KUKA KRL program: ps_ltc_geo_c2_Bolha.src, ps_ltc_geo_c2_Bolha.dat

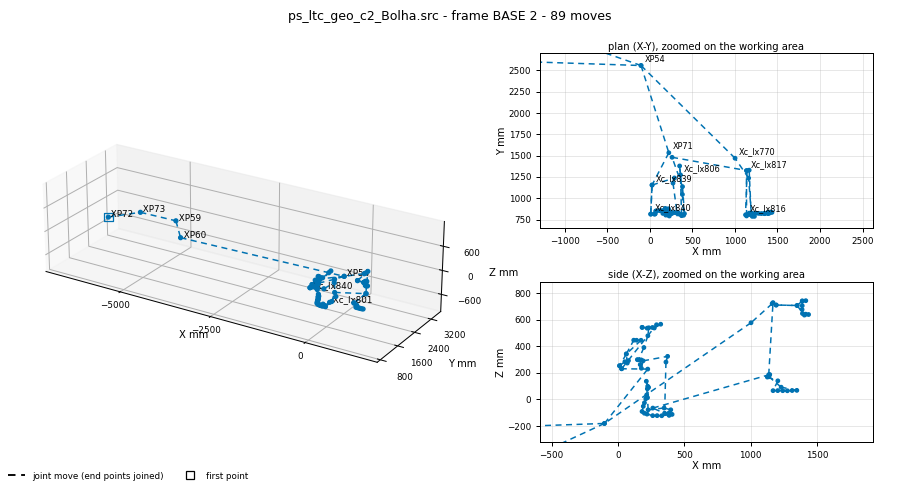
[picture p0: tool path of ps_ltc_geo_c2_Bolha.src in frame BASE 2, 89 of 89 moves have a stored position in this frame; points joined in program order, loops and branches not executed]
--- ps_ltc_geo_c2_Bolha.src ---
&ACCESS RVO1
&REL 11
&COMMENT Solda GUN C2 Geometria
&PARAM DISKPATH = KRC:\R1\Program\SOLDA LTC
DEF ps_ltc_geo_c2_Bolha( )
;FOLD INI
;FOLD SPOTTECH INI
USERSPOT(#INIT)
;ENDFOLD (SPOTTECH INI)
  ;FOLD USER INI
    ;Make your modifications here

  ;ENDFOLD (USER INI)
;ENDFOLD (INI)

; Caracterização dos meios de produção:
; Versão Atual: 03/11/2017
; Changes: Accelo Bolha
; Name: P13.050-R4


chk_w2_wechs_ok ( )     ; CHECK FERRAMENTA: C2

if MaxStandMenge (2) then
  MaxStandmengeErreicht (2)
endif

IF (NOT(GHOST())) THEN
if Elektrodenwechsel (2) then
  e_fraes2()
endif
ENDIF

;FOLD PTP P72 Vel=100 % PDAT95 Tool[2]:GUN C2 Base[2]:ACCELO;%{PE}%R 8.2.20,%MKUKATPBASIS,%CMOVE,%VPTP,%P 1:PTP, 2:P72, 3:, 5:100, 7:PDAT95
$BWDSTART=FALSE
PDAT_ACT=PPDAT95
FDAT_ACT=FP72
BAS(#PTP_PARAMS,100)
PTP XP72
;ENDFOLD
;FOLD PTP P73 CONT Vel=100 % PDAT96 Tool[2]:GUN C2 Base[2]:ACCELO;%{PE}%R 8.2.20,%MKUKATPBASIS,%CMOVE,%VPTP,%P 1:PTP, 2:P73, 3:C_DIS, 5:100, 7:PDAT96
$BWDSTART=FALSE
PDAT_ACT=PPDAT96
FDAT_ACT=FP73
BAS(#PTP_PARAMS,100)
PTP XP73 C_DIS
;ENDFOLD
;FOLD PTP P59 CONT Vel=100 % PDAT79 Tool[2]:GUN C2 Base[2]:ACCELO;%{PE}%R 8.2.20,%MKUKATPBASIS,%CMOVE,%VPTP,%P 1:PTP, 2:P59, 3:C_DIS, 5:100, 7:PDAT79
$BWDSTART=FALSE
PDAT_ACT=PPDAT79
FDAT_ACT=FP59
BAS(#PTP_PARAMS,100)
PTP XP59 C_DIS
;ENDFOLD
;FOLD PTP P60 CONT Vel=100 % PDAT80 Tool[2]:GUN C2 Base[2]:ACCELO;%{PE}%R 8.2.20,%MKUKATPBASIS,%CMOVE,%VPTP,%P 1:PTP, 2:P60, 3:C_DIS, 5:100, 7:PDAT80
$BWDSTART=FALSE
PDAT_ACT=PPDAT80
FDAT_ACT=FP60
BAS(#PTP_PARAMS,100)
PTP XP60 C_DIS
;ENDFOLD
;FOLD PTP P54 CONT Vel=100 % PDAT74 Tool[2]:GUN C2 Base[2]:ACCELO;%{PE}%R 8.2.20,%MKUKATPBASIS,%CMOVE,%VPTP,%P 1:PTP, 2:P54, 3:C_DIS, 5:100, 7:PDAT74
$BWDSTART=FALSE
PDAT_ACT=PPDAT74
FDAT_ACT=FP54
BAS(#PTP_PARAMS,100)
PTP XP54 C_DIS
;ENDFOLD


;FOLD OUT 3339 'R4 soldando' State=TRUE ;%{PE}%R 8.2.20,%MKUKATPBASIS,%COUT,%VOUTX,%P 2:3339, 3:R4 soldando, 5:TRUE, 6:
$OUT[3339]=TRUE
;ENDFOLD
;FOLD WAIT FOR ( IN 3339 'Aguarda lib solsar geometria' );%{PE}%R 8.2.20,%MKUKATPBASIS,%CEXT_WAIT_FOR,%VEXT_WAIT_FOR,%P 2:, 4:, 5:$IN, 6:3339, 7:Aguarda lib solsar geometria, 9:
WAIT FOR  ( $IN[3339] )
;ENDFOLD
;FOLD OUT 3339 'R4 soldando' State=FALSE ;%{PE}%R 8.2.20,%MKUKATPBASIS,%COUT,%VOUTX,%P 2:3339, 3:R4 soldando, 5:FALSE, 6:
$OUT[3339]=FALSE
;ENDFOLD
;FOLD OUT 3348 'Fora area GEOBOX' State=FALSE ;%{PE}%R 8.2.20,%MKUKATPBASIS,%COUT,%VOUTX,%P 2:3348, 3:Fora area GEOBOX, 5:FALSE, 6:
$OUT[3348]=FALSE
;ENDFOLD

;FOLD Collision.Monitoring_AREA_2_On ;%{PE}%MKUKATPUSER
COLLSTOP( 8, 1 ) ;not Interrupt-Controlled
;ENDFOLD


;FOLD PTP P71 CONT Vel=100 % PDAT94 Tool[2]:GUN C2 Base[2]:ACCELO;%{PE}%R 8.2.20,%MKUKATPBASIS,%CMOVE,%VPTP,%P 1:PTP, 2:P71, 3:C_DIS, 5:100, 7:PDAT94
$BWDSTART=FALSE
PDAT_ACT=PPDAT94
FDAT_ACT=FP71
BAS(#PTP_PARAMS,100)
PTP XP71 C_DIS
;ENDFOLD
;FOLD PTP c_lx839 CONT Vel=100 % P_OLP100 Tool[2]:GUN C2 Base[2]:ACCELO;%{PE}%R 8.2.20,%MKUKATPBASIS,%CMOVE,%VPTP,%P 1:PTP, 2:c_lx839, 3:C_DIS, 5:100, 7:P_OLP100
$BWDSTART=FALSE
PDAT_ACT=PP_OLP100
FDAT_ACT=Fc_lx839
BAS(#PTP_PARAMS,100)
PTP Xc_lx839 C_DIS
;ENDFOLD
;FOLD PTP c_lx840 CONT Vel=100 % P_OLP101 Tool[2]:GUN C2 Base[2]:ACCELO;%{PE}%R 8.2.20,%MKUKATPBASIS,%CMOVE,%VPTP,%P 1:PTP, 2:c_lx840, 3:C_DIS, 5:100, 7:P_OLP101
$BWDSTART=FALSE
PDAT_ACT=PP_OLP101
FDAT_ACT=Fc_lx840
BAS(#PTP_PARAMS,100)
PTP Xc_lx840 C_DIS
;ENDFOLD
;FOLD PTP P61 CONT Vel=100 % PDAT81 Tool[2]:GUN C2 Base[2]:ACCELO;%{PE}%R 8.2.20,%MKUKATPBASIS,%CMOVE,%VPTP,%P 1:PTP, 2:P61, 3:C_DIS, 5:100, 7:PDAT81
$BWDSTART=FALSE
PDAT_ACT=PPDAT81
FDAT_ACT=FP61
BAS(#PTP_PARAMS,100)
PTP XP61 C_DIS
;ENDFOLD

;FOLD ; swp_60_0220;%{PE}%R 8.2.20,%MKUKATPBASIS,%CCOMMENT,%VNORMAL,%P 2:swp_60_0220
;ENDFOLD
;FOLD PTP swp_60_0220 PDAT82 SPOT Gun=2 RETR CLS PGNO1=111 ACTIVE=1 Tool[2]:GUN C2 Base[2]:ACCELO;%{PE}%R 8.2.2,%MKUKATPSPOT,%CSPOT,%VPTP,%P 1:PTP, 2:swp_60_0220, 3:, 5:100, 7:PDAT82, 10:2, 12:#FIRST, 14:#CLO, 16:152, 18:1, 20:1, 22:0, 24:1, 25:S_OLP2
$BWDSTART=FALSE
PDAT_ACT=PPDAT82
FDAT_ACT=Fswp_60_0220
BAS(#PTP_PARAMS,PPDAT82.VEL)
S_ACT.GUN=2
S_ACT.PAIR=SDEFAULT.PAIR
S_ACT.RETR=#CLO
S_ACT.CLO_TM=1
S_ACT.PGNO1=111
S_ACT.PGNO2=SDEFAULT.PGNO2
S_ACT.PRESS1=SDEFAULT.PRESS1
S_ACT.PRESS2=SDEFAULT.PRESS2
S_READY=FALSE
PTP Xswp_60_0220
USERSPOT(#SPOT, S_ACT)
WAIT FOR S_READY
;ENDFOLD

;FOLD ; swp_60_0218;%{PE}%R 8.2.20,%MKUKATPBASIS,%CCOMMENT,%VNORMAL,%P 2:swp_60_0218
;ENDFOLD
;FOLD PTP swp_60_0218 PDAT83 SPOT Gun=2 RETR OPN PGNO1=112 ACTIVE=1 Tool[2]:GUN C2 Base[2]:ACCELO;%{PE}%R 8.2.2,%MKUKATPSPOT,%CSPOT,%VPTP,%P 1:PTP, 2:swp_60_0218, 3:, 5:100, 7:PDAT83, 10:2, 12:#FIRST, 14:#OPN, 16:153, 18:1, 20:1, 22:0, 24:1, 25:S_OLP3
$BWDSTART=FALSE
PDAT_ACT=PPDAT83
FDAT_ACT=Fswp_60_0218
BAS(#PTP_PARAMS,PPDAT83.VEL)
S_ACT.GUN=2
S_ACT.PAIR=SDEFAULT.PAIR
S_ACT.RETR=#OPN
S_ACT.CLO_TM=1
S_ACT.PGNO1=112
S_ACT.PGNO2=SDEFAULT.PGNO2
S_ACT.PRESS1=SDEFAULT.PRESS1
S_ACT.PRESS2=SDEFAULT.PRESS2
S_READY=FALSE
PTP Xswp_60_0218
USERSPOT(#SPOT, S_ACT)
WAIT FOR S_READY
;ENDFOLD

;FOLD PTP P62 CONT Vel=100 % PDAT84 Tool[2]:GUN C2 Base[2]:ACCELO;%{PE}%R 8.2.20,%MKUKATPBASIS,%CMOVE,%VPTP,%P 1:PTP, 2:P62, 3:C_DIS, 5:100, 7:PDAT84
$BWDSTART=FALSE
PDAT_ACT=PPDAT84
FDAT_ACT=FP62
BAS(#PTP_PARAMS,100)
PTP XP62 C_DIS
;ENDFOLD

;FOLD ; swp_60_0212;%{PE}%R 8.2.20,%MKUKATPBASIS,%CCOMMENT,%VNORMAL,%P 2:swp_60_0212
;ENDFOLD
;FOLD PTP swp_60_0212 PDAT85 SPOT Gun=2 RETR CLS PGNO1=109 ACTIVE=1 Tool[2]:GUN C2 Base[2]:ACCELO;%{PE}%R 8.2.2,%MKUKATPSPOT,%CSPOT,%VPTP,%P 1:PTP, 2:swp_60_0212, 3:, 5:100, 7:PDAT85, 10:2, 12:#FIRST, 14:#CLO, 16:150, 18:1, 20:0, 22:0, 24:1, 25:NORMAL
$BWDSTART=FALSE
PDAT_ACT=PPDAT85
FDAT_ACT=Fswp_60_0212
BAS(#PTP_PARAMS,PPDAT85.VEL)
S_ACT.GUN=2
S_ACT.PAIR=SDEFAULT.PAIR
S_ACT.RETR=#CLO
S_ACT.CLO_TM=1
S_ACT.PGNO1=109
S_ACT.PGNO2=SDEFAULT.PGNO2
S_ACT.PRESS1=SDEFAULT.PRESS1
S_ACT.PRESS2=SDEFAULT.PRESS2
S_READY=FALSE
PTP Xswp_60_0212
USERSPOT(#SPOT, S_ACT)
WAIT FOR S_READY
;ENDFOLD

;FOLD ; swp_60_0210;%{PE}%R 8.2.20,%MKUKATPBASIS,%CCOMMENT,%VNORMAL,%P 2:swp_60_0210
;ENDFOLD
;FOLD PTP swp_60_0210 PDAT86 SPOT Gun=2 RETR CLS PGNO1=113 ACTIVE=1 Tool[2]:GUN C2 Base[2]:ACCELO;%{PE}%R 8.2.2,%MKUKATPSPOT,%CSPOT,%VPTP,%P 1:PTP, 2:swp_60_0210, 3:, 5:100, 7:PDAT86, 10:2, 12:#FIRST, 14:#CLO, 16:154, 18:1, 20:1, 22:0, 24:1, 25:S_OLP4
$BWDSTART=FALSE
PDAT_ACT=PPDAT86
FDAT_ACT=Fswp_60_0210
BAS(#PTP_PARAMS,PPDAT86.VEL)
S_ACT.GUN=2
S_ACT.PAIR=SDEFAULT.PAIR
S_ACT.RETR=#CLO
S_ACT.CLO_TM=1
S_ACT.PGNO1=113
S_ACT.PGNO2=SDEFAULT.PGNO2
S_ACT.PRESS1=SDEFAULT.PRESS1
S_ACT.PRESS2=SDEFAULT.PRESS2
S_READY=FALSE
PTP Xswp_60_0210
USERSPOT(#SPOT, S_ACT)
WAIT FOR S_READY
;ENDFOLD

;FOLD ; swp_60_0208;%{PE}%R 8.2.20,%MKUKATPBASIS,%CCOMMENT,%VNORMAL,%P 2:swp_60_0208
;ENDFOLD
;FOLD PTP swp_60_0208 PDAT87 SPOT Gun=2 RETR OPN PGNO1=108 ACTIVE=1 Tool[2]:GUN C2 Base[2]:ACCELO;%{PE}%R 8.2.2,%MKUKATPSPOT,%CSPOT,%VPTP,%P 1:PTP, 2:swp_60_0208, 3:, 5:100, 7:PDAT87, 10:2, 12:#FIRST, 14:#OPN, 16:149, 18:1, 20:0, 22:0, 24:1, 25:NORMAL
$BWDSTART=FALSE
PDAT_ACT=PPDAT87
FDAT_ACT=Fswp_60_0208
BAS(#PTP_PARAMS,PPDAT87.VEL)
S_ACT.GUN=2
S_ACT.PAIR=SDEFAULT.PAIR
S_ACT.RETR=#OPN
S_ACT.CLO_TM=1
S_ACT.PGNO1=108
S_ACT.PGNO2=SDEFAULT.PGNO2
S_ACT.PRESS1=SDEFAULT.PRESS1
S_ACT.PRESS2=SDEFAULT.PRESS2
S_READY=FALSE
PTP Xswp_60_0208
USERSPOT(#SPOT, S_ACT)
WAIT FOR S_READY
;ENDFOLD

;FOLD PTP P65 CONT Vel=100 % PDAT88 Tool[2]:GUN C2 Base[2]:ACCELO;%{PE}%R 8.2.20,%MKUKATPBASIS,%CMOVE,%VPTP,%P 1:PTP, 2:P65, 3:C_DIS, 5:100, 7:PDAT88
$BWDSTART=FALSE
PDAT_ACT=PPDAT88
FDAT_ACT=FP65
BAS(#PTP_PARAMS,100)
PTP XP65 C_DIS
;ENDFOLD
;FOLD PTP P66 CONT Vel=100 % PDAT89 Tool[2]:GUN C2 Base[2]:ACCELO;%{PE}%R 8.2.20,%MKUKATPBASIS,%CMOVE,%VPTP,%P 1:PTP, 2:P66, 3:C_DIS, 5:100, 7:PDAT89
$BWDSTART=FALSE
PDAT_ACT=PPDAT89
FDAT_ACT=FP66
BAS(#PTP_PARAMS,100)
PTP XP66 C_DIS
;ENDFOLD
;FOLD PTP P67 CONT Vel=100 % PDAT90 Tool[2]:GUN C2 Base[2]:ACCELO;%{PE}%R 8.2.20,%MKUKATPBASIS,%CMOVE,%VPTP,%P 1:PTP, 2:P67, 3:C_DIS, 5:100, 7:PDAT90
$BWDSTART=FALSE
PDAT_ACT=PPDAT90
FDAT_ACT=FP67
BAS(#PTP_PARAMS,100)
PTP XP67 C_DIS
;ENDFOLD
;FOLD PTP P68 CONT Vel=100 % PDAT91 Tool[2]:GUN C2 Base[2]:ACCELO;%{PE}%R 8.2.20,%MKUKATPBASIS,%CMOVE,%VPTP,%P 1:PTP, 2:P68, 3:C_DIS, 5:100, 7:PDAT91
$BWDSTART=FALSE
PDAT_ACT=PPDAT91
FDAT_ACT=FP68
BAS(#PTP_PARAMS,100)
PTP XP68 C_DIS
;ENDFOLD
;FOLD PTP P69 CONT Vel=100 % PDAT92 Tool[2]:GUN C2 Base[2]:ACCELO;%{PE}%R 8.2.20,%MKUKATPBASIS,%CMOVE,%VPTP,%P 1:PTP, 2:P69, 3:C_DIS, 5:100, 7:PDAT92
$BWDSTART=FALSE
PDAT_ACT=PPDAT92
FDAT_ACT=FP69
BAS(#PTP_PARAMS,100)
PTP XP69 C_DIS
;ENDFOLD
;FOLD PTP c_lx791 CONT Vel=100 % P_OLP29 Tool[2]:GUN C2 Base[2]:ACCELO;%{PE}%R8.2,%MKUKATPBASIS,%CMOVE,%VPTP,%P 1:PTP, 2:c_lx791, 3:C_DIS, 5:100, 7:P_OLP29
$BWDSTART = FALSE
PDAT_ACT= PP_OLP29
FDAT_ACT= Fc_lx791
BAS(#PTP_PARAMS,100)
PTP Xc_lx791 C_DIS
;ENDFOLD
;FOLD PTP c_lx794 CONT Vel=100 % P_OLP30 Tool[2]:GUN C2 Base[2]:ACCELO;%{PE}%R8.2,%MKUKATPBASIS,%CMOVE,%VPTP,%P 1:PTP, 2:c_lx794, 3:C_DIS, 5:100, 7:P_OLP30
$BWDSTART = FALSE
PDAT_ACT= PP_OLP30
FDAT_ACT= Fc_lx794
BAS(#PTP_PARAMS,100)
PTP Xc_lx794 C_DIS
;ENDFOLD
;FOLD PTP P10 CONT Vel=100 % PDAT19 Tool[2]:GUN C2 Base[2]:ACCELO;%{PE}%R 8.2.20,%MKUKATPBASIS,%CMOVE,%VPTP,%P 1:PTP, 2:P10, 3:C_DIS, 5:100, 7:PDAT19
$BWDSTART=FALSE
PDAT_ACT=PPDAT19
FDAT_ACT=FP10
BAS(#PTP_PARAMS,100)
PTP XP10 C_DIS
;ENDFOLD

;FOLD ; swp_60_0202;%{PE}%R 8.2.20,%MKUKATPBASIS,%CCOMMENT,%VNORMAL,%P 2:swp_60_0202
;ENDFOLD
;FOLD PTP swp_60_0202 PDAT29 SPOT Gun=2 RETR CLS PGNO1=110 ACTIVE=1 Tool[2]:GUN C2 Base[2]:ACCELO;%{PE}%R 8.2.2,%MKUKATPSPOT,%CSPOT,%VPTP,%P 1:PTP, 2:swp_60_0202, 3:, 5:100, 7:PDAT29, 10:2, 12:#FIRST, 14:#CLO, 16:151, 18:1, 20:1, 22:0, 24:1, 25:S_OLP1
$BWDSTART=FALSE
PDAT_ACT=PPDAT29
FDAT_ACT=Fswp_60_0202
BAS(#PTP_PARAMS,PPDAT29.VEL)
S_ACT.GUN=2
S_ACT.PAIR=SDEFAULT.PAIR
S_ACT.RETR=#CLO
S_ACT.CLO_TM=1
S_ACT.PGNO1=110
S_ACT.PGNO2=SDEFAULT.PGNO2
S_ACT.PRESS1=SDEFAULT.PRESS1
S_ACT.PRESS2=SDEFAULT.PRESS2
S_READY=FALSE
PTP Xswp_60_0202
USERSPOT(#SPOT, S_ACT)
WAIT FOR S_READY
;ENDFOLD

;FOLD ; swp 60_0204;%{PE}%R 8.2.20,%MKUKATPBASIS,%CCOMMENT,%VNORMAL,%P 2:swp  60_0204
;ENDFOLD
;FOLD PTP swp_60_0204 PDAT44 SPOT Gun=2 RETR OPN PgNo1=107 ACTIVE=1 Tool[2]:GUN C2 Base[2]:ACCELO;%{PE}%R 8.2.2,%MKUKATPSPOT,%CSPOT,%VPTP,%P 1:PTP, 2:swp_60_0204, 3:, 5:100, 7:PDAT44, 10:2, 12:#FIRST, 14:#OPN, 16:107, 18:1, 20:0, 22:0, 24:1, 25:NORMAL
$BWDSTART=FALSE
PDAT_ACT=PPDAT44
FDAT_ACT=Fswp_60_0204
BAS(#PTP_PARAMS,PPDAT44.VEL)
S_ACT.GUN=2
S_ACT.PAIR=SDEFAULT.PAIR
S_ACT.RETR=#OPN
S_ACT.CLO_TM=1
S_ACT.PGNO1=107
S_ACT.PGNO2=SDEFAULT.PGNO2
S_ACT.PRESS1=SDEFAULT.PRESS1
S_ACT.PRESS2=SDEFAULT.PRESS2
S_READY=FALSE
PTP Xswp_60_0204
USERSPOT(#SPOT, S_ACT)
WAIT FOR S_READY
;ENDFOLD

;FOLD PTP P28 CONT Vel=100 % PDAT45 Tool[2]:GUN C2 Base[2]:ACCELO;%{PE}%R 8.2.20,%MKUKATPBASIS,%CMOVE,%VPTP,%P 1:PTP, 2:P28, 3:C_DIS, 5:100, 7:PDAT45
$BWDSTART=FALSE
PDAT_ACT=PPDAT45
FDAT_ACT=FP28
BAS(#PTP_PARAMS,100)
PTP XP28 C_DIS
;ENDFOLD

;FOLD ; swp_60_0206;%{PE}%R 8.2.20,%MKUKATPBASIS,%CCOMMENT,%VNORMAL,%P 2:swp_60_0206
;ENDFOLD
;FOLD PTP swp_60_0206 P_OLP92 SPOT Gun=2 RETR OPN PGNO1=114 ACTIVE=1 Tool[2]:GUN C2 Base[2]:ACCELO;%{PE}%R 8.2.2,%MKUKATPSPOT,%CSPOT,%VPTP,%P 1:PTP, 2:swp_60_0206, 3:, 5:100, 7:P_OLP92, 10:2, 12:#FIRST, 14:#OPN, 16:155, 18:1, 20:1, 22:0, 24:1, 25:S_OLP5
$BWDSTART=FALSE
PDAT_ACT=PP_OLP92
FDAT_ACT=Fswp_60_0206
BAS(#PTP_PARAMS,PP_OLP92.VEL)
S_ACT.GUN=2
S_ACT.PAIR=SDEFAULT.PAIR
S_ACT.RETR=#OPN
S_ACT.CLO_TM=1
S_ACT.PGNO1=114
S_ACT.PGNO2=SDEFAULT.PGNO2
S_ACT.PRESS1=SDEFAULT.PRESS1
S_ACT.PRESS2=SDEFAULT.PRESS2
S_READY=FALSE
PTP Xswp_60_0206
USERSPOT(#SPOT, S_ACT)
WAIT FOR S_READY
;ENDFOLD

;FOLD PTP c_lx836 CONT Vel=100 % P_OLP93 Tool[2]:GUN C2 Base[2]:ACCELO;%{PE}%R 8.2.20,%MKUKATPBASIS,%CMOVE,%VPTP,%P 1:PTP, 2:c_lx836, 3:C_DIS, 5:100, 7:P_OLP93
$BWDSTART=FALSE
PDAT_ACT=PP_OLP93
FDAT_ACT=Fc_lx836
BAS(#PTP_PARAMS,100)
PTP Xc_lx836 C_DIS
;ENDFOLD
;FOLD PTP c_lx837 CONT Vel=100 % P_OLP94 Tool[2]:GUN C2 Base[2]:ACCELO;%{PE}%R 8.2.20,%MKUKATPBASIS,%CMOVE,%VPTP,%P 1:PTP, 2:c_lx837, 3:C_DIS, 5:100, 7:P_OLP94
$BWDSTART=FALSE
PDAT_ACT=PP_OLP94
FDAT_ACT=Fc_lx837
BAS(#PTP_PARAMS,100)
PTP Xc_lx837 C_DIS
;ENDFOLD

;FOLD ; swp_60_0222;%{PE}%R 8.2.20,%MKUKATPBASIS,%CCOMMENT,%VNORMAL,%P 2:swp_60_0222
;ENDFOLD
;FOLD PTP swp_60_0222 P_OLP95 SPOT Gun=2 RETR CLS PGNO1=115 ACTIVE=1 Tool[2]:GUN C2 Base[2]:ACCELO;%{PE}%R 8.2.2,%MKUKATPSPOT,%CSPOT,%VPTP,%P 1:PTP, 2:swp_60_0222, 3:, 5:100, 7:P_OLP95, 10:2, 12:#FIRST, 14:#CLO, 16:156, 18:1, 20:1, 22:0, 24:1, 25:S_OLP6
$BWDSTART=FALSE
PDAT_ACT=PP_OLP95
FDAT_ACT=Fswp_60_0222
BAS(#PTP_PARAMS,PP_OLP95.VEL)
S_ACT.GUN=2
S_ACT.PAIR=SDEFAULT.PAIR
S_ACT.RETR=#CLO
S_ACT.CLO_TM=1
S_ACT.PGNO1=115
S_ACT.PGNO2=SDEFAULT.PGNO2
S_ACT.PRESS1=SDEFAULT.PRESS1
S_ACT.PRESS2=SDEFAULT.PRESS2
S_READY=FALSE
PTP Xswp_60_0222
USERSPOT(#SPOT, S_ACT)
WAIT FOR S_READY
;ENDFOLD

;FOLD PTP c_lx838 CONT Vel=100 % P_OLP96 Tool[2]:GUN C2 Base[2]:ACCELO;%{PE}%R 8.2.20,%MKUKATPBASIS,%CMOVE,%VPTP,%P 1:PTP, 2:c_lx838, 3:C_DIS, 5:100, 7:P_OLP96
$BWDSTART=FALSE
PDAT_ACT=PP_OLP96
FDAT_ACT=Fc_lx838
BAS(#PTP_PARAMS,100)
PTP Xc_lx838 C_DIS
;ENDFOLD

;FOLD ; swp_60_0226;%{PE}%R 8.2.20,%MKUKATPBASIS,%CCOMMENT,%VNORMAL,%P 2:swp_60_0226
;ENDFOLD
;FOLD PTP swp_60_0226 P_OLP97 SPOT Gun=2 RETR CLS PGNO1=116 ACTIVE=1 Tool[2]:GUN C2 Base[2]:ACCELO;%{PE}%R 8.2.2,%MKUKATPSPOT,%CSPOT,%VPTP,%P 1:PTP, 2:swp_60_0226, 3:, 5:100, 7:P_OLP97, 10:2, 12:#FIRST, 14:#CLO, 16:157, 18:1, 20:1, 22:0, 24:1, 25:S_OLP7
$BWDSTART=FALSE
PDAT_ACT=PP_OLP97
FDAT_ACT=Fswp_60_0226
BAS(#PTP_PARAMS,PP_OLP97.VEL)
S_ACT.GUN=2
S_ACT.PAIR=SDEFAULT.PAIR
S_ACT.RETR=#CLO
S_ACT.CLO_TM=1
S_ACT.PGNO1=116
S_ACT.PGNO2=SDEFAULT.PGNO2
S_ACT.PRESS1=SDEFAULT.PRESS1
S_ACT.PRESS2=SDEFAULT.PRESS2
S_READY=FALSE
PTP Xswp_60_0226
USERSPOT(#SPOT, S_ACT)
WAIT FOR S_READY
;ENDFOLD

;FOLD ; swp_60_0230;%{PE}%R 5.4.33,%MKUKATPBASIS,%CCOMMENT,%VNORMAL,%P 2:swp_60_0230
;ENDFOLD
;FOLD PTP swp_60_0230 P_OLP38 SPOT Gun=2 RETR OPN PGNO1=117 ACTIVE=1 Tool[2]:GUN C2 Base[2]:ACCELO;%{PE}%R 8.2.2,%MKUKATPSPOT,%CSPOT,%VPTP,%P 1:PTP, 2:swp_60_0230, 3:, 5:100, 7:P_OLP38, 10:2, 12:#FIRST, 14:#OPN, 16:158, 18:1, 20:1, 22:0, 24:1, 25:S_OLP8
$BWDSTART=FALSE
PDAT_ACT=PP_OLP38
FDAT_ACT=Fswp_60_0230
BAS(#PTP_PARAMS,PP_OLP38.VEL)
S_ACT.GUN=2
S_ACT.PAIR=SDEFAULT.PAIR
S_ACT.RETR=#OPN
S_ACT.CLO_TM=1
S_ACT.PGNO1=117
S_ACT.PGNO2=SDEFAULT.PGNO2
S_ACT.PRESS1=SDEFAULT.PRESS1
S_ACT.PRESS2=SDEFAULT.PRESS2
S_READY=FALSE
PTP Xswp_60_0230
USERSPOT(#SPOT, S_ACT)
WAIT FOR S_READY
;ENDFOLD

;FOLD PTP c_lx803 CONT Vel=100 % P_OLP39 Tool[2]:GUN C2 Base[2]:ACCELO;%{PE}%R8.2,%MKUKATPBASIS,%CMOVE,%VPTP,%P 1:PTP, 2:c_lx803, 3:C_DIS, 5:100, 7:P_OLP39
$BWDSTART = FALSE
PDAT_ACT= PP_OLP39
FDAT_ACT= Fc_lx803
BAS(#PTP_PARAMS,100)
PTP Xc_lx803 C_DIS
;ENDFOLD
;FOLD PTP P26 CONT Vel=100 % PDAT43 Tool[2]:GUN C2 Base[2]:ACCELO;%{PE}%R 8.2.20,%MKUKATPBASIS,%CMOVE,%VPTP,%P 1:PTP, 2:P26, 3:C_DIS, 5:100, 7:PDAT43
$BWDSTART=FALSE
PDAT_ACT=PPDAT43
FDAT_ACT=FP26
BAS(#PTP_PARAMS,100)
PTP XP26 C_DIS
;ENDFOLD
;FOLD PTP c_lx806 CONT Vel=100 % P_OLP42 Tool[2]:GUN C2 Base[2]:ACCELO;%{PE}%R8.2,%MKUKATPBASIS,%CMOVE,%VPTP,%P 1:PTP, 2:c_lx806, 3:C_DIS, 5:100, 7:P_OLP42
$BWDSTART = FALSE
PDAT_ACT= PP_OLP42
FDAT_ACT= Fc_lx806
BAS(#PTP_PARAMS,100)
PTP Xc_lx806 C_DIS
;ENDFOLD
;FOLD PTP c_lx831 Vel=100 % P_OLP86 Tool[2]:GUN C2 Base[2]:ACCELO;%{PE}%R 8.2.20,%MKUKATPBASIS,%CMOVE,%VPTP,%P 1:PTP, 2:c_lx831, 3:, 5:100, 7:P_OLP86
$BWDSTART=FALSE
PDAT_ACT=PP_OLP86
FDAT_ACT=Fc_lx831
BAS(#PTP_PARAMS,100)
PTP Xc_lx831
;ENDFOLD
;FOLD PTP c_lx801 CONT Vel=100 % P_OLP46 Tool[2]:GUN C2 Base[2]:ACCELO;%{PE}%R 8.2.20,%MKUKATPBASIS,%CMOVE,%VPTP,%P 1:PTP, 2:c_lx801, 3:C_DIS, 5:100, 7:P_OLP46
$BWDSTART=FALSE
PDAT_ACT=PP_OLP46
FDAT_ACT=Fc_lx801
BAS(#PTP_PARAMS,100)
PTP Xc_lx801 C_DIS
;ENDFOLD
;FOLD PTP c_lx802 CONT Vel=100 % P_OLP47 Tool[2]:GUN C2 Base[2]:ACCELO;%{PE}%R 8.2.20,%MKUKATPBASIS,%CMOVE,%VPTP,%P 1:PTP, 2:c_lx802, 3:C_DIS, 5:100, 7:P_OLP47
$BWDSTART=FALSE
PDAT_ACT=PP_OLP47
FDAT_ACT=Fc_lx802
BAS(#PTP_PARAMS,100)
PTP Xc_lx802 C_DIS
;ENDFOLD
;FOLD PTP c_lx800 CONT Vel=100 % P_OLP48 Tool[2]:GUN C2 Base[2]:ACCELO;%{PE}%R 8.2.20,%MKUKATPBASIS,%CMOVE,%VPTP,%P 1:PTP, 2:c_lx800, 3:C_DIS, 5:100, 7:P_OLP48
$BWDSTART=FALSE
PDAT_ACT=PP_OLP48
FDAT_ACT=Fc_lx800
BAS(#PTP_PARAMS,100)
PTP Xc_lx800 C_DIS
;ENDFOLD
;FOLD PTP c_lx799 CONT Vel=100 % P_OLP49 Tool[2]:GUN C2 Base[2]:ACCELO;%{PE}%R 8.2.20,%MKUKATPBASIS,%CMOVE,%VPTP,%P 1:PTP, 2:c_lx799, 3:C_DIS, 5:100, 7:P_OLP49
$BWDSTART=FALSE
PDAT_ACT=PP_OLP49
FDAT_ACT=Fc_lx799
BAS(#PTP_PARAMS,100)
PTP Xc_lx799 C_DIS
;ENDFOLD
;FOLD PTP P7 CONT Vel=100 % PDAT16 Tool[2]:GUN C2 Base[2]:ACCELO;%{PE}%R 8.2.20,%MKUKATPBASIS,%CMOVE,%VPTP,%P 1:PTP, 2:P7, 3:C_DIS, 5:100, 7:PDAT16
$BWDSTART=FALSE
PDAT_ACT=PPDAT16
FDAT_ACT=FP7
BAS(#PTP_PARAMS,100)
PTP XP7 C_DIS
;ENDFOLD
;FOLD PTP c_lx798 CONT Vel=100 % P_OLP50 Tool[2]:GUN C2 Base[2]:ACCELO;%{PE}%R 8.2.20,%MKUKATPBASIS,%CMOVE,%VPTP,%P 1:PTP, 2:c_lx798, 3:C_DIS, 5:100, 7:P_OLP50
$BWDSTART=FALSE
PDAT_ACT=PP_OLP50
FDAT_ACT=Fc_lx798
BAS(#PTP_PARAMS,100)
PTP Xc_lx798 C_DIS
;ENDFOLD

;FOLD ; swp_60_0236;%{PE}%R 5.4.33,%MKUKATPBASIS,%CCOMMENT,%VNORMAL,%P 2:swp_60_0236
;ENDFOLD
;FOLD PTP swp_60_0236 P_OLP51 SPOT Gun=2 RETR CLS PGNO1=118 ACTIVE=1 Tool[2]:GUN C2 Base[2]:ACCELO;%{PE}%R 8.2.2,%MKUKATPSPOT,%CSPOT,%VPTP,%P 1:PTP, 2:swp_60_0236, 3:, 5:100, 7:P_OLP51, 10:2, 12:#FIRST, 14:#CLO, 16:159, 18:1, 20:1, 22:0, 24:1, 25:S_OLP9
$BWDSTART=FALSE
PDAT_ACT=PP_OLP51
FDAT_ACT=Fswp_60_0236
BAS(#PTP_PARAMS,PP_OLP51.VEL)
S_ACT.GUN=2
S_ACT.PAIR=SDEFAULT.PAIR
S_ACT.RETR=#CLO
S_ACT.CLO_TM=1
S_ACT.PGNO1=118
S_ACT.PGNO2=SDEFAULT.PGNO2
S_ACT.PRESS1=SDEFAULT.PRESS1
S_ACT.PRESS2=SDEFAULT.PRESS2
S_READY=FALSE
PTP Xswp_60_0236
USERSPOT(#SPOT, S_ACT)
WAIT FOR S_READY
;ENDFOLD

;FOLD ; swp_60_0238;%{PE}%R 8.2.20,%MKUKATPBASIS,%CCOMMENT,%VNORMAL,%P 2:swp_60_0238
;ENDFOLD
;FOLD PTP swp_60_0238 PDAT63 SPOT Gun=2 RETR CLS PGNO1=102 ACTIVE=1 Tool[2]:GUN C2 Base[2]:ACCELO;%{PE}%R 8.2.2,%MKUKATPSPOT,%CSPOT,%VPTP,%P 1:PTP, 2:swp_60_0238, 3:, 5:100, 7:PDAT63, 10:2, 12:#FIRST, 14:#CLO, 16:143, 18:1, 20:0, 22:0, 24:1, 25:NORMAL
$BWDSTART=FALSE
PDAT_ACT=PPDAT63
FDAT_ACT=Fswp_60_0238
BAS(#PTP_PARAMS,PPDAT63.VEL)
S_ACT.GUN=2
S_ACT.PAIR=SDEFAULT.PAIR
S_ACT.RETR=#CLO
S_ACT.CLO_TM=1
S_ACT.PGNO1=102
S_ACT.PGNO2=SDEFAULT.PGNO2
S_ACT.PRESS1=SDEFAULT.PRESS1
S_ACT.PRESS2=SDEFAULT.PRESS2
S_READY=FALSE
PTP Xswp_60_0238
USERSPOT(#SPOT, S_ACT)
WAIT FOR S_READY
;ENDFOLD

;FOLD ; swp_60_0240;%{PE}%R 8.2.20,%MKUKATPBASIS,%CCOMMENT,%VNORMAL,%P 2:swp_60_0240
;ENDFOLD
;FOLD PTP swp_60_0240 PDAT64 SPOT Gun=2 RETR CLS PGNO1=101 ACTIVE=1 Tool[2]:GUN C2 Base[2]:ACCELO;%{PE}%R 8.2.2,%MKUKATPSPOT,%CSPOT,%VPTP,%P 1:PTP, 2:swp_60_0240, 3:, 5:100, 7:PDAT64, 10:2, 12:#FIRST, 14:#CLO, 16:142, 18:1, 20:0, 22:0, 24:1, 25:NORMAL
$BWDSTART=FALSE
PDAT_ACT=PPDAT64
FDAT_ACT=Fswp_60_0240
BAS(#PTP_PARAMS,PPDAT64.VEL)
S_ACT.GUN=2
S_ACT.PAIR=SDEFAULT.PAIR
S_ACT.RETR=#CLO
S_ACT.CLO_TM=1
S_ACT.PGNO1=101
S_ACT.PGNO2=SDEFAULT.PGNO2
S_ACT.PRESS1=SDEFAULT.PRESS1
S_ACT.PRESS2=SDEFAULT.PRESS2
S_READY=FALSE
PTP Xswp_60_0240
USERSPOT(#SPOT, S_ACT)
WAIT FOR S_READY
;ENDFOLD

;FOLD ; swp_60_0242;%{PE}%R 8.2.20,%MKUKATPBASIS,%CCOMMENT,%VNORMAL,%P 2:swp_60_0242
;ENDFOLD
;FOLD PTP swp_60_0242 PDAT65 SPOT Gun=2 RETR CLS PGNO1=100 ACTIVE=1 Tool[2]:GUN C2 Base[2]:ACCELO;%{PE}%R 8.2.2,%MKUKATPSPOT,%CSPOT,%VPTP,%P 1:PTP, 2:swp_60_0242, 3:, 5:100, 7:PDAT65, 10:2, 12:#FIRST, 14:#CLO, 16:141, 18:1, 20:0, 22:0, 24:1, 25:NORMAL
$BWDSTART=FALSE
PDAT_ACT=PPDAT65
FDAT_ACT=Fswp_60_0242
BAS(#PTP_PARAMS,PPDAT65.VEL)
S_ACT.GUN=2
S_ACT.PAIR=SDEFAULT.PAIR
S_ACT.RETR=#CLO
S_ACT.CLO_TM=1
S_ACT.PGNO1=100
S_ACT.PGNO2=SDEFAULT.PGNO2
S_ACT.PRESS1=SDEFAULT.PRESS1
S_ACT.PRESS2=SDEFAULT.PRESS2
S_READY=FALSE
PTP Xswp_60_0242
USERSPOT(#SPOT, S_ACT)
WAIT FOR S_READY
;ENDFOLD

;FOLD ; swp_60_0244;%{PE}%R 8.2.20,%MKUKATPBASIS,%CCOMMENT,%VNORMAL,%P 2:swp_60_0244
;ENDFOLD
;FOLD PTP swp_60_0244 PDAT66 SPOT Gun=2 RETR CLS PGNO1=99 ACTIVE=1 Tool[2]:GUN C2 Base[2]:ACCELO;%{PE}%R 8.2.2,%MKUKATPSPOT,%CSPOT,%VPTP,%P 1:PTP, 2:swp_60_0244, 3:, 5:100, 7:PDAT66, 10:2, 12:#FIRST, 14:#CLO, 16:140, 18:1, 20:0, 22:0, 24:1, 25:NORMAL
$BWDSTART=FALSE
PDAT_ACT=PPDAT66
FDAT_ACT=Fswp_60_0244
BAS(#PTP_PARAMS,PPDAT66.VEL)
S_ACT.GUN=2
S_ACT.PAIR=SDEFAULT.PAIR
S_ACT.RETR=#CLO
S_ACT.CLO_TM=1
S_ACT.PGNO1=99
S_ACT.PGNO2=SDEFAULT.PGNO2
S_ACT.PRESS1=SDEFAULT.PRESS1
S_ACT.PRESS2=SDEFAULT.PRESS2
S_READY=FALSE
PTP Xswp_60_0244
USERSPOT(#SPOT, S_ACT)
WAIT FOR S_READY
;ENDFOLD

;FOLD ; swp_60_0246;%{PE}%R 8.2.20,%MKUKATPBASIS,%CCOMMENT,%VNORMAL,%P 2:swp_60_0246
;ENDFOLD
;FOLD PTP swp_60_0246 P_OLP98 SPOT Gun=2 RETR CLS PGNO1=119 ACTIVE=1 Tool[2]:GUN C2 Base[2]:ACCELO;%{PE}%R 8.2.2,%MKUKATPSPOT,%CSPOT,%VPTP,%P 1:PTP, 2:swp_60_0246, 3:, 5:100, 7:P_OLP98, 10:2, 12:#FIRST, 14:#CLO, 16:160, 18:1, 20:1, 22:0, 24:1, 25:S_OLP10
$BWDSTART=FALSE
PDAT_ACT=PP_OLP98
FDAT_ACT=Fswp_60_0246
BAS(#PTP_PARAMS,PP_OLP98.VEL)
S_ACT.GUN=2
S_ACT.PAIR=SDEFAULT.PAIR
S_ACT.RETR=#CLO
S_ACT.CLO_TM=1
S_ACT.PGNO1=119
S_ACT.PGNO2=SDEFAULT.PGNO2
S_ACT.PRESS1=SDEFAULT.PRESS1
S_ACT.PRESS2=SDEFAULT.PRESS2
S_READY=FALSE
PTP Xswp_60_0246
USERSPOT(#SPOT, S_ACT)
WAIT FOR S_READY
;ENDFOLD

;FOLD ; swp_60_0248;%{PE}%R 8.2.20,%MKUKATPBASIS,%CCOMMENT,%VNORMAL,%P 2:swp_60_0248
;ENDFOLD
;FOLD PTP swp_60_0248 PDAT67 SPOT Gun=2 RETR CLS PGNO1=98 ACTIVE=1 Tool[2]:GUN C2 Base[2]:ACCELO;%{PE}%R 8.2.2,%MKUKATPSPOT,%CSPOT,%VPTP,%P 1:PTP, 2:swp_60_0248, 3:, 5:100, 7:PDAT67, 10:2, 12:#FIRST, 14:#CLO, 16:139, 18:1, 20:0, 22:0, 24:1, 25:NORMAL
$BWDSTART=FALSE
PDAT_ACT=PPDAT67
FDAT_ACT=Fswp_60_0248
BAS(#PTP_PARAMS,PPDAT67.VEL)
S_ACT.GUN=2
S_ACT.PAIR=SDEFAULT.PAIR
S_ACT.RETR=#CLO
S_ACT.CLO_TM=1
S_ACT.PGNO1=98
S_ACT.PGNO2=SDEFAULT.PGNO2
S_ACT.PRESS1=SDEFAULT.PRESS1
S_ACT.PRESS2=SDEFAULT.PRESS2
S_READY=FALSE
PTP Xswp_60_0248
USERSPOT(#SPOT, S_ACT)
WAIT FOR S_READY
;ENDFOLD

;FOLD ; swp_60_0250;%{PE}%R 8.2.20,%MKUKATPBASIS,%CCOMMENT,%VNORMAL,%P 2:swp_60_0250
;ENDFOLD
;FOLD PTP swp_60_0250 PDAT68 SPOT Gun=2 RETR CLS PGNO1=97 ACTIVE=1 Tool[2]:GUN C2 Base[2]:ACCELO;%{PE}%R 8.2.2,%MKUKATPSPOT,%CSPOT,%VPTP,%P 1:PTP, 2:swp_60_0250, 3:, 5:100, 7:PDAT68, 10:2, 12:#FIRST, 14:#CLO, 16:138, 18:1, 20:0, 22:0, 24:1, 25:NORMAL
$BWDSTART=FALSE
PDAT_ACT=PPDAT68
FDAT_ACT=Fswp_60_0250
BAS(#PTP_PARAMS,PPDAT68.VEL)
S_ACT.GUN=2
S_ACT.PAIR=SDEFAULT.PAIR
S_ACT.RETR=#CLO
S_ACT.CLO_TM=1
S_ACT.PGNO1=97
S_ACT.PGNO2=SDEFAULT.PGNO2
S_ACT.PRESS1=SDEFAULT.PRESS1
S_ACT.PRESS2=SDEFAULT.PRESS2
S_READY=FALSE
PTP Xswp_60_0250
USERSPOT(#SPOT, S_ACT)
WAIT FOR S_READY
;ENDFOLD

;FOLD ; swp_60_0252;%{PE}%R 8.2.20,%MKUKATPBASIS,%CCOMMENT,%VNORMAL,%P 2:swp_60_0252
;ENDFOLD
;FOLD PTP swp_60_0252 PDAT69 SPOT Gun=2 RETR CLS PGNO1=96 ACTIVE=1 Tool[2]:GUN C2 Base[2]:ACCELO;%{PE}%R 8.2.2,%MKUKATPSPOT,%CSPOT,%VPTP,%P 1:PTP, 2:swp_60_0252, 3:, 5:100, 7:PDAT69, 10:2, 12:#FIRST, 14:#CLO, 16:137, 18:1, 20:0, 22:0, 24:1, 25:NORMAL
$BWDSTART=FALSE
PDAT_ACT=PPDAT69
FDAT_ACT=Fswp_60_0252
BAS(#PTP_PARAMS,PPDAT69.VEL)
S_ACT.GUN=2
S_ACT.PAIR=SDEFAULT.PAIR
S_ACT.RETR=#CLO
S_ACT.CLO_TM=1
S_ACT.PGNO1=96
S_ACT.PGNO2=SDEFAULT.PGNO2
S_ACT.PRESS1=SDEFAULT.PRESS1
S_ACT.PRESS2=SDEFAULT.PRESS2
S_READY=FALSE
PTP Xswp_60_0252
USERSPOT(#SPOT, S_ACT)
WAIT FOR S_READY
;ENDFOLD

;FOLD ; swp_60_0254;%{PE}%R 8.2.20,%MKUKATPBASIS,%CCOMMENT,%VNORMAL,%P 2:swp_60_0254
;ENDFOLD
;FOLD PTP swp_60_0254 PDAT70 SPOT Gun=2 RETR CLS PGNO1=95 ACTIVE=1 Tool[2]:GUN C2 Base[2]:ACCELO;%{PE}%R 8.2.2,%MKUKATPSPOT,%CSPOT,%VPTP,%P 1:PTP, 2:swp_60_0254, 3:, 5:100, 7:PDAT70, 10:2, 12:#FIRST, 14:#CLO, 16:136, 18:1, 20:0, 22:0, 24:1, 25:NORMAL
$BWDSTART=FALSE
PDAT_ACT=PPDAT70
FDAT_ACT=Fswp_60_0254
BAS(#PTP_PARAMS,PPDAT70.VEL)
S_ACT.GUN=2
S_ACT.PAIR=SDEFAULT.PAIR
S_ACT.RETR=#CLO
S_ACT.CLO_TM=1
S_ACT.PGNO1=95
S_ACT.PGNO2=SDEFAULT.PGNO2
S_ACT.PRESS1=SDEFAULT.PRESS1
S_ACT.PRESS2=SDEFAULT.PRESS2
S_READY=FALSE
PTP Xswp_60_0254
USERSPOT(#SPOT, S_ACT)
WAIT FOR S_READY
;ENDFOLD

;FOLD ; swp_60_0256;%{PE}%R 8.2.20,%MKUKATPBASIS,%CCOMMENT,%VNORMAL,%P 2:swp_60_0256
;ENDFOLD
;FOLD PTP swp_60_0256 P_OLP99 SPOT Gun=2 RETR CLS PGNO1=120 ACTIVE=1 Tool[2]:GUN C2 Base[2]:ACCELO;%{PE}%R 8.2.2,%MKUKATPSPOT,%CSPOT,%VPTP,%P 1:PTP, 2:swp_60_0256, 3:, 5:100, 7:P_OLP99, 10:2, 12:#FIRST, 14:#CLO, 16:161, 18:1, 20:1, 22:0, 24:1, 25:S_OLP11
$BWDSTART=FALSE
PDAT_ACT=PP_OLP99
FDAT_ACT=Fswp_60_0256
BAS(#PTP_PARAMS,PP_OLP99.VEL)
S_ACT.GUN=2
S_ACT.PAIR=SDEFAULT.PAIR
S_ACT.RETR=#CLO
S_ACT.CLO_TM=1
S_ACT.PGNO1=120
S_ACT.PGNO2=SDEFAULT.PGNO2
S_ACT.PRESS1=SDEFAULT.PRESS1
S_ACT.PRESS2=SDEFAULT.PRESS2
S_READY=FALSE
PTP Xswp_60_0256
USERSPOT(#SPOT, S_ACT)
WAIT FOR S_READY
;ENDFOLD

;FOLD ; swp_60_0258;%{PE}%R 8.2.20,%MKUKATPBASIS,%CCOMMENT,%VNORMAL,%P 2:swp_60_0258
;ENDFOLD
;FOLD PTP swp_60_0258 PDAT71 SPOT Gun=2 RETR CLS PGNO1=94 ACTIVE=1 Tool[2]:GUN C2 Base[2]:ACCELO;%{PE}%R 8.2.2,%MKUKATPSPOT,%CSPOT,%VPTP,%P 1:PTP, 2:swp_60_0258, 3:, 5:100, 7:PDAT71, 10:2, 12:#FIRST, 14:#CLO, 16:135, 18:1, 20:0, 22:0, 24:1, 25:NORMAL
$BWDSTART=FALSE
PDAT_ACT=PPDAT71
FDAT_ACT=Fswp_60_0258
BAS(#PTP_PARAMS,PPDAT71.VEL)
S_ACT.GUN=2
S_ACT.PAIR=SDEFAULT.PAIR
S_ACT.RETR=#CLO
S_ACT.CLO_TM=1
S_ACT.PGNO1=94
S_ACT.PGNO2=SDEFAULT.PGNO2
S_ACT.PRESS1=SDEFAULT.PRESS1
S_ACT.PRESS2=SDEFAULT.PRESS2
S_READY=FALSE
PTP Xswp_60_0258
USERSPOT(#SPOT, S_ACT)
WAIT FOR S_READY
;ENDFOLD

;FOLD ; swp_60_0260;%{PE}%R 8.2.20,%MKUKATPBASIS,%CCOMMENT,%VNORMAL,%P 2:swp_60_0260
;ENDFOLD
;FOLD PTP swp_60_0260 PDAT72 SPOT Gun=2 RETR OPN PGNO1=93 ACTIVE=1 Tool[2]:GUN C2 Base[2]:ACCELO;%{PE}%R 8.2.2,%MKUKATPSPOT,%CSPOT,%VPTP,%P 1:PTP, 2:swp_60_0260, 3:, 5:100, 7:PDAT72, 10:2, 12:#FIRST, 14:#OPN, 16:134, 18:1, 20:0, 22:0, 24:1, 25:NORMAL
$BWDSTART=FALSE
PDAT_ACT=PPDAT72
FDAT_ACT=Fswp_60_0260
BAS(#PTP_PARAMS,PPDAT72.VEL)
S_ACT.GUN=2
S_ACT.PAIR=SDEFAULT.PAIR
S_ACT.RETR=#OPN
S_ACT.CLO_TM=1
S_ACT.PGNO1=93
S_ACT.PGNO2=SDEFAULT.PGNO2
S_ACT.PRESS1=SDEFAULT.PRESS1
S_ACT.PRESS2=SDEFAULT.PRESS2
S_READY=FALSE
PTP Xswp_60_0260
USERSPOT(#SPOT, S_ACT)
WAIT FOR S_READY
;ENDFOLD

;FOLD PTP c_lx813 CONT Vel=100 % P_OLP57 Tool[2]:GUN C2 Base[2]:ACCELO;%{PE}%R 8.2.20,%MKUKATPBASIS,%CMOVE,%VPTP,%P 1:PTP, 2:c_lx813, 3:C_DIS, 5:100, 7:P_OLP57
$BWDSTART=FALSE
PDAT_ACT=PP_OLP57
FDAT_ACT=Fc_lx813
BAS(#PTP_PARAMS,100)
PTP Xc_lx813 C_DIS
;ENDFOLD
;FOLD PTP c_lx832 CONT Vel=100 % P_OLP88 Tool[2]:GUN C2 Base[2]:ACCELO;%{PE}%R 8.2.20,%MKUKATPBASIS,%CMOVE,%VPTP,%P 1:PTP, 2:c_lx832, 3:C_DIS, 5:100, 7:P_OLP88
$BWDSTART=FALSE
PDAT_ACT=PP_OLP88
FDAT_ACT=Fc_lx832
BAS(#PTP_PARAMS,100)
PTP Xc_lx832 C_DIS
;ENDFOLD
;FOLD PTP c_lx814 Vel=100 % P_OLP58 Tool[2]:GUN C2 Base[2]:ACCELO;%{PE}%R 8.2.20,%MKUKATPBASIS,%CMOVE,%VPTP,%P 1:PTP, 2:c_lx814, 3:, 5:100, 7:P_OLP58
$BWDSTART=FALSE
PDAT_ACT=PP_OLP58
FDAT_ACT=Fc_lx814
BAS(#PTP_PARAMS,100)
PTP Xc_lx814
;ENDFOLD


;FOLD Collision.Monitoring_AREA_3_On ;%{PE}%MKUKATPUSER
COLLSTOP( 9, 1 ) ;not Interrupt-Controlled
;ENDFOLD


;FOLD PTP c_lx817 CONT Vel=100 % P_OLP59 Tool[2]:GUN C2 Base[2]:ACCELO;%{PE}%R 8.2.20,%MKUKATPBASIS,%CMOVE,%VPTP,%P 1:PTP, 2:c_lx817, 3:C_DIS, 5:100, 7:P_OLP59
$BWDSTART=FALSE
PDAT_ACT=PP_OLP59
FDAT_ACT=Fc_lx817
BAS(#PTP_PARAMS,100)
PTP Xc_lx817 C_DIS
;ENDFOLD
;FOLD PTP c_lx816 CONT Vel=100 % P_OLP60 Tool[2]:GUN C2 Base[2]:ACCELO;%{PE}%R 8.2.20,%MKUKATPBASIS,%CMOVE,%VPTP,%P 1:PTP, 2:c_lx816, 3:C_DIS, 5:100, 7:P_OLP60
$BWDSTART=FALSE
PDAT_ACT=PP_OLP60
FDAT_ACT=Fc_lx816
BAS(#PTP_PARAMS,100)
PTP Xc_lx816 C_DIS
;ENDFOLD
;FOLD PTP c_lx815 CONT Vel=100 % P_OLP61 Tool[2]:GUN C2 Base[2]:ACCELO;%{PE}%R 8.2.20,%MKUKATPBASIS,%CMOVE,%VPTP,%P 1:PTP, 2:c_lx815, 3:C_DIS, 5:100, 7:P_OLP61
$BWDSTART=FALSE
PDAT_ACT=PP_OLP61
FDAT_ACT=Fc_lx815
BAS(#PTP_PARAMS,100)
PTP Xc_lx815 C_DIS
;ENDFOLD

;FOLD ; swp_0332;%{PE}%R 8.2.20,%MKUKATPBASIS,%CCOMMENT,%VNORMAL,%P 2:swp_0332
;ENDFOLD
;FOLD PTP swp_60_0332 P_OLP102 SPOT Gun=2 RETR CLS PGNO1=91 ACTIVE=1 Tool[2]:GUN C2 Base[2]:ACCELO;%{PE}%R 8.2.2,%MKUKATPSPOT,%CSPOT,%VPTP,%P 1:PTP, 2:swp_60_0332, 3:, 5:100, 7:P_OLP102, 10:2, 12:#FIRST, 14:#CLO, 16:132, 18:1, 20:1, 22:0, 24:1, 25:S_OLP12
$BWDSTART=FALSE
PDAT_ACT=PP_OLP102
FDAT_ACT=Fswp_60_0332
BAS(#PTP_PARAMS,PP_OLP102.VEL)
S_ACT.GUN=2
S_ACT.PAIR=SDEFAULT.PAIR
S_ACT.RETR=#CLO
S_ACT.CLO_TM=1
S_ACT.PGNO1=91
S_ACT.PGNO2=SDEFAULT.PGNO2
S_ACT.PRESS1=SDEFAULT.PRESS1
S_ACT.PRESS2=SDEFAULT.PRESS2
S_READY=FALSE
PTP Xswp_60_0332
USERSPOT(#SPOT, S_ACT)
WAIT FOR S_READY
;ENDFOLD

;FOLD ; swp_0334;%{PE}%R 8.2.20,%MKUKATPBASIS,%CCOMMENT,%VNORMAL,%P 2:swp_0334
;ENDFOLD
;FOLD PTP swp_60_0334 P_OLP62 SPOT Gun=2 RETR CLS PGNO1=121 ACTIVE=1 Tool[2]:GUN C2 Base[2]:ACCELO;%{PE}%R 8.2.2,%MKUKATPSPOT,%CSPOT,%VPTP,%P 1:PTP, 2:swp_60_0334, 3:, 5:100, 7:P_OLP62, 10:2, 12:#FIRST, 14:#CLO, 16:162, 18:1, 20:1, 22:0, 24:1, 25:S_OLP12
$BWDSTART=FALSE
PDAT_ACT=PP_OLP62
FDAT_ACT=Fswp_60_0334
BAS(#PTP_PARAMS,PP_OLP62.VEL)
S_ACT.GUN=2
S_ACT.PAIR=SDEFAULT.PAIR
S_ACT.RETR=#CLO
S_ACT.CLO_TM=1
S_ACT.PGNO1=121
S_ACT.PGNO2=SDEFAULT.PGNO2
S_ACT.PRESS1=SDEFAULT.PRESS1
S_ACT.PRESS2=SDEFAULT.PRESS2
S_READY=FALSE
PTP Xswp_60_0334
USERSPOT(#SPOT, S_ACT)
WAIT FOR S_READY
;ENDFOLD

;FOLD ; swp_0336;%{PE}%R 8.2.20,%MKUKATPBASIS,%CCOMMENT,%VNORMAL,%P 2:swp_0336
;ENDFOLD
;FOLD PTP swp_60_0336 P_OLP103 SPOT Gun=2 RETR CLS PGNO1=90 ACTIVE=1 Tool[2]:GUN C2 Base[2]:ACCELO;%{PE}%R 8.2.2,%MKUKATPSPOT,%CSPOT,%VPTP,%P 1:PTP, 2:swp_60_0336, 3:, 5:100, 7:P_OLP103, 10:2, 12:#FIRST, 14:#CLO, 16:131, 18:1, 20:1, 22:0, 24:1, 25:S_OLP12
$BWDSTART=FALSE
PDAT_ACT=PP_OLP103
FDAT_ACT=Fswp_60_0336
BAS(#PTP_PARAMS,PP_OLP103.VEL)
S_ACT.GUN=2
S_ACT.PAIR=SDEFAULT.PAIR
S_ACT.RETR=#CLO
S_ACT.CLO_TM=1
S_ACT.PGNO1=90
S_ACT.PGNO2=SDEFAULT.PGNO2
S_ACT.PRESS1=SDEFAULT.PRESS1
S_ACT.PRESS2=SDEFAULT.PRESS2
S_READY=FALSE
PTP Xswp_60_0336
USERSPOT(#SPOT, S_ACT)
WAIT FOR S_READY
;ENDFOLD


;FOLD Collision.Monitoring_AREA_1_On ;%{PE}%MKUKATPUSER
COLLSTOP( 7, 1 ) ;not Interrupt-Controlled
;ENDFOLD


;FOLD ; swp_0338;%{PE}%R 8.2.20,%MKUKATPBASIS,%CCOMMENT,%VNORMAL,%P 2:swp_0338
;ENDFOLD
;FOLD PTP swp_60_0338 P_OLP104 SPOT Gun=2 RETR CLS PGNO1=89 ACTIVE=1 Tool[2]:GUN C2 Base[2]:ACCELO;%{PE}%R 8.2.2,%MKUKATPSPOT,%CSPOT,%VPTP,%P 1:PTP, 2:swp_60_0338, 3:, 5:100, 7:P_OLP104, 10:2, 12:#FIRST, 14:#CLO, 16:130, 18:1, 20:1, 22:0, 24:1, 25:S_OLP12
$BWDSTART=FALSE
PDAT_ACT=PP_OLP104
FDAT_ACT=Fswp_60_0338
BAS(#PTP_PARAMS,PP_OLP104.VEL)
S_ACT.GUN=2
S_ACT.PAIR=SDEFAULT.PAIR
S_ACT.RETR=#CLO
S_ACT.CLO_TM=1
S_ACT.PGNO1=89
S_ACT.PGNO2=SDEFAULT.PGNO2
S_ACT.PRESS1=SDEFAULT.PRESS1
S_ACT.PRESS2=SDEFAULT.PRESS2
S_READY=FALSE
PTP Xswp_60_0338
USERSPOT(#SPOT, S_ACT)
WAIT FOR S_READY
;ENDFOLD

;FOLD ; swp_0340;%{PE}%R 8.2.20,%MKUKATPBASIS,%CCOMMENT,%VNORMAL,%P 2:swp_0340
;ENDFOLD
;FOLD PTP swp_60_0340 P_OLP105 SPOT Gun=2 RETR CLS PGNO1=88 ACTIVE=1 Tool[2]:GUN C2 Base[2]:ACCELO;%{PE}%R 8.2.2,%MKUKATPSPOT,%CSPOT,%VPTP,%P 1:PTP, 2:swp_60_0340, 3:, 5:100, 7:P_OLP105, 10:2, 12:#FIRST, 14:#CLO, 16:129, 18:1, 20:1, 22:0, 24:1, 25:S_OLP12
$BWDSTART=FALSE
PDAT_ACT=PP_OLP105
FDAT_ACT=Fswp_60_0340
BAS(#PTP_PARAMS,PP_OLP105.VEL)
S_ACT.GUN=2
S_ACT.PAIR=SDEFAULT.PAIR
S_ACT.RETR=#CLO
S_ACT.CLO_TM=1
S_ACT.PGNO1=88
S_ACT.PGNO2=SDEFAULT.PGNO2
S_ACT.PRESS1=SDEFAULT.PRESS1
S_ACT.PRESS2=SDEFAULT.PRESS2
S_READY=FALSE
PTP Xswp_60_0340
USERSPOT(#SPOT, S_ACT)
WAIT FOR S_READY
;ENDFOLD

;FOLD ; swp_60_0342;%{PE}%R 8.2.20,%MKUKATPBASIS,%CCOMMENT,%VNORMAL,%P 2:swp_60_0342
;ENDFOLD
;FOLD PTP swp_60_0342 P_OLP63 SPOT Gun=2 RETR OPN PGNO1=122 ACTIVE=1 Tool[2]:GUN C2 Base[2]:ACCELO;%{PE}%R 8.2.2,%MKUKATPSPOT,%CSPOT,%VPTP,%P 1:PTP, 2:swp_60_0342, 3:, 5:100, 7:P_OLP63, 10:2, 12:#FIRST, 14:#OPN, 16:163, 18:1, 20:1, 22:0, 24:1, 25:S_OLP13
$BWDSTART=FALSE
PDAT_ACT=PP_OLP63
FDAT_ACT=Fswp_60_0342
BAS(#PTP_PARAMS,PP_OLP63.VEL)
S_ACT.GUN=2
S_ACT.PAIR=SDEFAULT.PAIR
S_ACT.RETR=#OPN
S_ACT.CLO_TM=1
S_ACT.PGNO1=122
S_ACT.PGNO2=SDEFAULT.PGNO2
S_ACT.PRESS1=SDEFAULT.PRESS1
S_ACT.PRESS2=SDEFAULT.PRESS2
S_READY=FALSE
PTP Xswp_60_0342
USERSPOT(#SPOT, S_ACT)
WAIT FOR S_READY
;ENDFOLD

;FOLD PTP c_lx820 CONT Vel=100 % P_OLP66 Tool[2]:GUN C2 Base[2]:ACCELO;%{PE}%R 8.2.20,%MKUKATPBASIS,%CMOVE,%VPTP,%P 1:PTP, 2:c_lx820, 3:C_DIS, 5:100, 7:P_OLP66
$BWDSTART=FALSE
PDAT_ACT=PP_OLP66
FDAT_ACT=Fc_lx820
BAS(#PTP_PARAMS,100)
PTP Xc_lx820 C_DIS
;ENDFOLD
;FOLD PTP P3 CONT Vel=100 % PDAT3 Tool[2]:GUN C2 Base[2]:ACCELO;%{PE}%R 8.2.20,%MKUKATPBASIS,%CMOVE,%VPTP,%P 1:PTP, 2:P3, 3:C_DIS, 5:100, 7:PDAT3
$BWDSTART=FALSE
PDAT_ACT=PPDAT3
FDAT_ACT=FP3
BAS(#PTP_PARAMS,100)
PTP XP3 C_DIS
;ENDFOLD
;FOLD PTP P22 CONT Vel=100 % PDAT38 Tool[2]:GUN C2 Base[2]:ACCELO;%{PE}%R 8.2.20,%MKUKATPBASIS,%CMOVE,%VPTP,%P 1:PTP, 2:P22, 3:C_DIS, 5:100, 7:PDAT38
$BWDSTART=FALSE
PDAT_ACT=PPDAT38
FDAT_ACT=FP22
BAS(#PTP_PARAMS,100)
PTP XP22 C_DIS
;ENDFOLD
;FOLD PTP c_lx822 CONT Vel=100 % P_OLP67 Tool[2]:GUN C2 Base[2]:ACCELO;%{PE}%R 8.2.20,%MKUKATPBASIS,%CMOVE,%VPTP,%P 1:PTP, 2:c_lx822, 3:C_DIS, 5:100, 7:P_OLP67
$BWDSTART=FALSE
PDAT_ACT=PP_OLP67
FDAT_ACT=Fc_lx822
BAS(#PTP_PARAMS,100)
PTP Xc_lx822 C_DIS
;ENDFOLD


;FOLD Collision.Monitoring_AREA_4_On ;%{PE}%MKUKATPUSER
COLLSTOP( 10, 1 ) ;not Interrupt-Controlled
;ENDFOLD


;FOLD PTP c_lx823 CONT Vel=100 % P_OLP68 Tool[2]:GUN C2 Base[2]:ACCELO;%{PE}%R 8.2.20,%MKUKATPBASIS,%CMOVE,%VPTP,%P 1:PTP, 2:c_lx823, 3:C_DIS, 5:100, 7:P_OLP68
$BWDSTART=FALSE
PDAT_ACT=PP_OLP68
FDAT_ACT=Fc_lx823
BAS(#PTP_PARAMS,100)
PTP Xc_lx823 C_DIS
;ENDFOLD
;FOLD PTP c_lx821 CONT Vel=100 % P_OLP69 Tool[2]:GUN C2 Base[2]:ACCELO;%{PE}%R 8.2.20,%MKUKATPBASIS,%CMOVE,%VPTP,%P 1:PTP, 2:c_lx821, 3:C_DIS, 5:100, 7:P_OLP69
$BWDSTART=FALSE
PDAT_ACT=PP_OLP69
FDAT_ACT=Fc_lx821
BAS(#PTP_PARAMS,100)
PTP Xc_lx821 C_DIS
;ENDFOLD
;FOLD PTP P24 CONT Vel=100 % PDAT41 Tool[2]:GUN C2 Base[2]:ACCELO;%{PE}%R 8.2.20,%MKUKATPBASIS,%CMOVE,%VPTP,%P 1:PTP, 2:P24, 3:C_DIS, 5:100, 7:PDAT41
$BWDSTART=FALSE
PDAT_ACT=PPDAT41
FDAT_ACT=FP24
BAS(#PTP_PARAMS,100)
PTP XP24 C_DIS
;ENDFOLD

;FOLD ; swp_60_0392n;%{PE}%R 8.2.20,%MKUKATPBASIS,%CCOMMENT,%VNORMAL,%P 2:swp_60_0392n
;ENDFOLD
;FOLD PTP swp_60_0392 P_OLP77 SPOT Gun=2 RETR CLS PgNo1=141 ACTIVE=1 Tool[2]:GUN C2 Base[2]:ACCELO;%{PE}%R 8.2.2,%MKUKATPSPOT,%CSPOT,%VPTP,%P 1:PTP, 2:swp_60_0392, 3:, 5:100, 7:P_OLP77, 10:2, 12:#FIRST, 14:#CLO, 16:141, 18:1, 20:1, 22:0, 24:1, 25:S_OLP14
$BWDSTART=FALSE
PDAT_ACT=PP_OLP77
FDAT_ACT=Fswp_60_0392
BAS(#PTP_PARAMS,PP_OLP77.VEL)
S_ACT.GUN=2
S_ACT.PAIR=SDEFAULT.PAIR
S_ACT.RETR=#CLO
S_ACT.CLO_TM=1
S_ACT.PGNO1=141
S_ACT.PGNO2=SDEFAULT.PGNO2
S_ACT.PRESS1=SDEFAULT.PRESS1
S_ACT.PRESS2=SDEFAULT.PRESS2
S_READY=FALSE
PTP Xswp_60_0392
USERSPOT(#SPOT, S_ACT)
WAIT FOR S_READY
;ENDFOLD

;FOLD ; swp_60_0394;%{PE}%R 5.4.33,%MKUKATPBASIS,%CCOMMENT,%VNORMAL,%P 2:swp_60_0394
;ENDFOLD
;FOLD PTP swp_60_0394 P_OLP70 SPOT Gun=2 RETR CLS PgNo1=124 ACTIVE=1 Tool[2]:GUN C2 Base[2]:ACCELO;%{PE}%R 8.2.2,%MKUKATPSPOT,%CSPOT,%VPTP,%P 1:PTP, 2:swp_60_0394, 3:, 5:100, 7:P_OLP70, 10:2, 12:#FIRST, 14:#CLO, 16:124, 18:1, 20:1, 22:0, 24:1, 25:S_OLP14
$BWDSTART=FALSE
PDAT_ACT=PP_OLP70
FDAT_ACT=Fswp_60_0394
BAS(#PTP_PARAMS,PP_OLP70.VEL)
S_ACT.GUN=2
S_ACT.PAIR=SDEFAULT.PAIR
S_ACT.RETR=#CLO
S_ACT.CLO_TM=1
S_ACT.PGNO1=124
S_ACT.PGNO2=SDEFAULT.PGNO2
S_ACT.PRESS1=SDEFAULT.PRESS1
S_ACT.PRESS2=SDEFAULT.PRESS2
S_READY=FALSE
PTP Xswp_60_0394
USERSPOT(#SPOT, S_ACT)
WAIT FOR S_READY
;ENDFOLD

;FOLD PTP c_lx824 CONT Vel=100 % P_OLP71 Tool[2]:GUN C2 Base[2]:ACCELO;%{PE}%R 8.2.20,%MKUKATPBASIS,%CMOVE,%VPTP,%P 1:PTP, 2:c_lx824, 3:C_DIS, 5:100, 7:P_OLP71
$BWDSTART=FALSE
PDAT_ACT=PP_OLP71
FDAT_ACT=Fc_lx824
BAS(#PTP_PARAMS,100)
PTP Xc_lx824 C_DIS
;ENDFOLD

;FOLD ; swp_60_0396;%{PE}%R 5.4.33,%MKUKATPBASIS,%CCOMMENT,%VNORMAL,%P 2:swp_60_0396
;ENDFOLD
;FOLD PTP swp_60_0396 P_OLP72 SPOT Gun=2 RETR CLS PGNO1=124 ACTIVE=1 Tool[2]:GUN C2 Base[2]:ACCELO;%{PE}%R 8.2.2,%MKUKATPSPOT,%CSPOT,%VPTP,%P 1:PTP, 2:swp_60_0396, 3:, 5:100, 7:P_OLP72, 10:2, 12:#FIRST, 14:#CLO, 16:165, 18:1, 20:1, 22:0, 24:1, 25:S_OLP15
$BWDSTART=FALSE
PDAT_ACT=PP_OLP72
FDAT_ACT=Fswp_60_0396
BAS(#PTP_PARAMS,PP_OLP72.VEL)
S_ACT.GUN=2
S_ACT.PAIR=SDEFAULT.PAIR
S_ACT.RETR=#CLO
S_ACT.CLO_TM=1
S_ACT.PGNO1=124
S_ACT.PGNO2=SDEFAULT.PGNO2
S_ACT.PRESS1=SDEFAULT.PRESS1
S_ACT.PRESS2=SDEFAULT.PRESS2
S_READY=FALSE
PTP Xswp_60_0396
USERSPOT(#SPOT, S_ACT)
WAIT FOR S_READY
;ENDFOLD

;FOLD ; swp_60_0398n;%{PE}%R 8.2.20,%MKUKATPBASIS,%CCOMMENT,%VNORMAL,%P 2:swp_60_0398n
;ENDFOLD
;FOLD PTP swp_60_0398 P_OLP81 SPOT Gun=2 RETR CLS PgNo1=140 ACTIVE=1 Tool[2]:GUN C2 Base[2]:ACCELO;%{PE}%R 8.2.2,%MKUKATPSPOT,%CSPOT,%VPTP,%P 1:PTP, 2:swp_60_0398, 3:, 5:100, 7:P_OLP81, 10:2, 12:#FIRST, 14:#CLO, 16:140, 18:1, 20:1, 22:0, 24:1, 25:S_OLP15
$BWDSTART=FALSE
PDAT_ACT=PP_OLP81
FDAT_ACT=Fswp_60_0398
BAS(#PTP_PARAMS,PP_OLP81.VEL)
S_ACT.GUN=2
S_ACT.PAIR=SDEFAULT.PAIR
S_ACT.RETR=#CLO
S_ACT.CLO_TM=1
S_ACT.PGNO1=140
S_ACT.PGNO2=SDEFAULT.PGNO2
S_ACT.PRESS1=SDEFAULT.PRESS1
S_ACT.PRESS2=SDEFAULT.PRESS2
S_READY=FALSE
PTP Xswp_60_0398
USERSPOT(#SPOT, S_ACT)
WAIT FOR S_READY
;ENDFOLD

;FOLD PTP c_lx825 CONT Vel=100 % P_OLP73 Tool[2]:GUN C2 Base[2]:ACCELO;%{PE}%R 8.2.20,%MKUKATPBASIS,%CMOVE,%VPTP,%P 1:PTP, 2:c_lx825, 3:C_DIS, 5:100, 7:P_OLP73
$BWDSTART=FALSE
PDAT_ACT=PP_OLP73
FDAT_ACT=Fc_lx825
BAS(#PTP_PARAMS,100)
PTP Xc_lx825 C_DIS
;ENDFOLD

;FOLD ; swp_60_0400;%{PE}%R 5.4.33,%MKUKATPBASIS,%CCOMMENT,%VNORMAL,%P 2:swp_60_0400
;ENDFOLD
;FOLD PTP swp_60_0400 P_OLP74 SPOT Gun=2 RETR OPN PgNo1=124 ACTIVE=1 Tool[2]:GUN C2 Base[2]:ACCELO;%{PE}%R 8.2.2,%MKUKATPSPOT,%CSPOT,%VPTP,%P 1:PTP, 2:swp_60_0400, 3:, 5:100, 7:P_OLP74, 10:2, 12:#FIRST, 14:#OPN, 16:124, 18:1, 20:1, 22:0, 24:1, 25:S_OLP16
$BWDSTART=FALSE
PDAT_ACT=PP_OLP74
FDAT_ACT=Fswp_60_0400
BAS(#PTP_PARAMS,PP_OLP74.VEL)
S_ACT.GUN=2
S_ACT.PAIR=SDEFAULT.PAIR
S_ACT.RETR=#OPN
S_ACT.CLO_TM=1
S_ACT.PGNO1=124
S_ACT.PGNO2=SDEFAULT.PGNO2
S_ACT.PRESS1=SDEFAULT.PRESS1
S_ACT.PRESS2=SDEFAULT.PRESS2
S_READY=FALSE
PTP Xswp_60_0400
USERSPOT(#SPOT, S_ACT)
WAIT FOR S_READY
;ENDFOLD

;FOLD PTP c_lx826 CONT Vel=100 % P_OLP75 Tool[2]:GUN C2 Base[2]:ACCELO;%{PE}%R 8.2.20,%MKUKATPBASIS,%CMOVE,%VPTP,%P 1:PTP, 2:c_lx826, 3:C_DIS, 5:100, 7:P_OLP75
$BWDSTART=FALSE
PDAT_ACT=PP_OLP75
FDAT_ACT=Fc_lx826
BAS(#PTP_PARAMS,100)
PTP Xc_lx826 C_DIS
;ENDFOLD
;FOLD PTP c_lx827 CONT Vel=100 % P_OLP76 Tool[2]:GUN C2 Base[2]:ACCELO;%{PE}%R 8.2.20,%MKUKATPBASIS,%CMOVE,%VPTP,%P 1:PTP, 2:c_lx827, 3:C_DIS, 5:100, 7:P_OLP76
$BWDSTART=FALSE
PDAT_ACT=PP_OLP76
FDAT_ACT=Fc_lx827
BAS(#PTP_PARAMS,100)
PTP Xc_lx827 C_DIS
;ENDFOLD
;FOLD PTP c_lx829 CONT Vel=100 % P_OLP78 Tool[2]:GUN C2 Base[2]:ACCELO;%{PE}%R 8.2.20,%MKUKATPBASIS,%CMOVE,%VPTP,%P 1:PTP, 2:c_lx829, 3:C_DIS, 5:100, 7:P_OLP78
$BWDSTART=FALSE
PDAT_ACT=PP_OLP78
FDAT_ACT=Fc_lx829
BAS(#PTP_PARAMS,100)
PTP Xc_lx829 C_DIS
;ENDFOLD


;FOLD Collision.Monitoring_AREA_4_Off . ;%{PE}%MKUKATPUSER
COLLSTOP( 10, 2+0 )
;ENDFOLD


;FOLD PTP c_lx830 CONT Vel=100 % P_OLP79 Tool[2]:GUN C2 Base[2]:ACCELO;%{PE}%R 8.2.20,%MKUKATPBASIS,%CMOVE,%VPTP,%P 1:PTP, 2:c_lx830, 3:C_DIS, 5:100, 7:P_OLP79
$BWDSTART=FALSE
PDAT_ACT=PP_OLP79
FDAT_ACT=Fc_lx830
BAS(#PTP_PARAMS,100)
PTP Xc_lx830 C_DIS
;ENDFOLD
;FOLD PTP c_lx770 CONT Vel=100 % P_OLP80 Tool[2]:GUN C2 Base[2]:ACCELO;%{PE}%R 8.2.20,%MKUKATPBASIS,%CMOVE,%VPTP,%P 1:PTP, 2:c_lx770, 3:C_DIS, 5:100, 7:P_OLP80
$BWDSTART=FALSE
PDAT_ACT=PP_OLP80
FDAT_ACT=Fc_lx770
BAS(#PTP_PARAMS,100)
PTP Xc_lx770 C_DIS
;ENDFOLD
;FOLD PTP P57 CONT Vel=100 % PDAT77 Tool[2]:GUN C2 Base[2]:ACCELO;%{PE}%R 8.2.20,%MKUKATPBASIS,%CMOVE,%VPTP,%P 1:PTP, 2:P57, 3:C_DIS, 5:100, 7:PDAT77
$BWDSTART=FALSE
PDAT_ACT=PPDAT77
FDAT_ACT=FP57
BAS(#PTP_PARAMS,100)
PTP XP57 C_DIS
;ENDFOLD


;FOLD Collision.Monitoring_AREA_3_Off . ;%{PE}%MKUKATPUSER
COLLSTOP( 9, 2+0 )
;ENDFOLD
;FOLD Collision.Monitoring_AREA_2_Off . ;%{PE}%MKUKATPUSER
COLLSTOP( 8, 2+0 )
;ENDFOLD
;FOLD Collision.Monitoring_AREA_1_Off . ;%{PE}%MKUKATPUSER
COLLSTOP( 7, 2+0 )
;ENDFOLD


;FOLD PTP P53 CONT Vel=100 % PDAT73 Tool[2]:GUN C2 Base[2]:ACCELO;%{PE}%R 8.2.20,%MKUKATPBASIS,%CMOVE,%VPTP,%P 1:PTP, 2:P53, 3:C_DIS, 5:100, 7:PDAT73
$BWDSTART=FALSE
PDAT_ACT=PPDAT73
FDAT_ACT=FP53
BAS(#PTP_PARAMS,100)
PTP XP53 C_DIS
;ENDFOLD


end_weld_GEO()           ; Bit fim solda geometria

;FOLD OUT 3348 'Fora area GEOBOX' State=TRUE ;%{PE}%R 8.2.20,%MKUKATPBASIS,%COUT,%VOUTX,%P 2:3348, 3:Fora area GEOBOX, 5:TRUE, 6:
$OUT[3348]=TRUE
;ENDFOLD


END

--- ps_ltc_geo_c2_Bolha.dat ---
&ACCESS RVO1
&REL 11
&COMMENT Solda GUN C2 Geometria
&PARAM DISKPATH = KRC:\R1\Program\SOLDA LTC
DEFDAT  ps_ltc_geo_c2_Bolha
;FOLD EXTERNAL DECLARATIONS;%{PE}%MKUKATPBASIS,%CEXT,%VCOMMON,%P
;FOLD GRIPPERTECH EXT
EXT  H50 (INT  :IN,INT  :IN,INT  :IN,GRP_TYP  :IN )
;ENDFOLD (GRIPPERTECH EXT)
;FOLD SPOTTECH EXT
EXT  USERSPOT (S_COMMAND  :IN,SPOT_TYPE  :IN )
;ENDFOLD (SPOTTECH EXT)
;FOLD BASISTECH EXT;%{PE}%MKUKATPBASIS,%CEXT,%VEXT,%P
EXT  BAS (BAS_COMMAND  :IN,REAL  :IN )
DECL INT SUCCESS
;ENDFOLD (BASISTECH EXT)
;FOLD USER EXT;%{E}%MKUKATPUSER,%CEXT,%VEXT,%P
;Make your modifications here

;ENDFOLD (USER EXT)
;ENDFOLD (EXTERNAL DECLARATIONS)

;# ============ START PATH : swp_p13050r4_ltc_geo_c2 =============
DECL FDAT Fswp_60_0202={TOOL_NO 2,BASE_NO 2,IPO_FRAME #BASE,POINT2[] " "}
DECL SPOT_TYPE SS_OLP1={GUN 1,PAIR #FIRST,RETR #OPN,CLO_TM 0,PGNO1 1,PRESS1 1.0,PGNO2 0,PRESS2 0.0}
DECL E6POS Xswp_60_0202={X 182.835007,Y 880.438416,Z 543.002197,A 178.139694,B -18.2308292,C 93.6574173,S 2,T 34,E1 5325.16992,E2 0.0,E3 0.0,E4 0.0,E5 0.0,E6 0.0}
DECL FDAT Fswp_60_0220={TOOL_NO 2,BASE_NO 2,IPO_FRAME #BASE,POINT2[] " "}
DECL SPOT_TYPE SS_OLP2={GUN 1,PAIR #FIRST,RETR #OPN,CLO_TM 0,PGNO1 1,PRESS1 1.0,PGNO2 0,PRESS2 0.0}
DECL E6POS Xswp_60_0220={X 78.6135101,Y 851.181885,Z 292.565491,A -8.68553352,B -28.2226295,C -89.2399979,S 2,T 2,E1 5234.21289,E2 0.0,E3 0.0,E4 0.0,E5 0.0,E6 0.0}
DECL FDAT Fswp_60_0218={TOOL_NO 2,BASE_NO 2,IPO_FRAME #BASE,POINT2[] " "}
DECL SPOT_TYPE SS_OLP3={GUN 1,PAIR #FIRST,RETR #OPN,CLO_TM 0,PGNO1 1,PRESS1 1.0,PGNO2 0,PRESS2 0.0}
DECL E6POS Xswp_60_0218={X 69.8426666,Y 849.211487,Z 274.013611,A -15.2370596,B -27.2786102,C -83.9252701,S 2,T 2,E1 5234.21582,E2 0.0,E3 0.0,E4 0.0,E5 0.0,E6 0.0}
DECL FDAT Fswp_60_0210={TOOL_NO 2,BASE_NO 2,IPO_FRAME #BASE,POINT2[] " "}
DECL SPOT_TYPE SS_OLP4={GUN 1,PAIR #FIRST,RETR #OPN,CLO_TM 0,PGNO1 1,PRESS1 1.0,PGNO2 0,PRESS2 0.0}
DECL E6POS Xswp_60_0210={X 139.787094,Y 852.099426,Z 445.815186,A 2.35583401,B -46.1486702,C -94.2666016,S 2,T 2,E1 5234.42578,E2 0.0,E3 0.0,E4 0.0,E5 0.0,E6 0.0}
DECL FDAT Fc_lx791={TOOL_NO 2,BASE_NO 2,IPO_FRAME #BASE,POINT2[] " "}
DECL PDAT PP_OLP29={VEL 100.0,ACC 100.0,APO_DIST 100.0,APO_MODE #CDIS}
DECL E6POS Xc_lx791={X 321.637695,Y 822.888794,Z 566.796387,A -175.408203,B -36.04039,C 92.2376404,S 2,T 2,E1 5325.1748,E2 0.0,E3 0.0,E4 0.0,E5 0.0,E6 0.0}
DECL FDAT Fc_lx794={TOOL_NO 2,BASE_NO 2,IPO_FRAME #BASE,POINT2[] " "}
DECL PDAT PP_OLP30={VEL 100.0,ACC 100.0,APO_DIST 100.0,APO_MODE #CDIS}
DECL E6POS Xc_lx794={X 259.54071,Y 819.94458,Z 542.128723,A -174.497299,B -26.6495705,C 92.4456177,S 2,T 2,E1 5325.17383,E2 0.0,E3 0.0,E4 0.0,E5 0.0,E6 0.0}
DECL FDAT Fswp_60_0206={TOOL_NO 2,BASE_NO 2,IPO_FRAME #BASE,POINT2[] " "}
DECL SPOT_TYPE SS_OLP5={GUN 1,PAIR #FIRST,RETR #OPN,CLO_TM 0,PGNO1 1,PRESS1 1.0,PGNO2 0,PRESS2 0.0}
DECL E6POS Xswp_60_0206={X 224.979202,Y 854.995911,Z 479.702209,A 178.734497,B -6.96247816,C 91.0636368,S 2,T 34,E1 5346.75488,E2 0.0,E3 0.0,E4 0.0,E5 0.0,E6 0.0}
DECL FDAT Fswp_60_0222={TOOL_NO 2,BASE_NO 2,IPO_FRAME #BASE,POINT2[] " "}
DECL SPOT_TYPE SS_OLP6={GUN 1,PAIR #FIRST,RETR #OPN,CLO_TM 0,PGNO1 1,PRESS1 1.0,PGNO2 0,PRESS2 0.0}
DECL E6POS Xswp_60_0222={X 145.817505,Y 851.460815,Z 300.019897,A 176.8246,B 14.5630703,C 87.8208466,S 2,T 34,E1 5341.86377,E2 0.0,E3 0.0,E4 0.0,E5 0.0,E6 0.0}
DECL FDAT Fswp_60_0226={TOOL_NO 2,BASE_NO 2,IPO_FRAME #BASE,POINT2[] " "}
DECL SPOT_TYPE SS_OLP7={GUN 1,PAIR #FIRST,RETR #OPN,CLO_TM 0,PGNO1 1,PRESS1 1.0,PGNO2 0,PRESS2 0.0}
DECL E6POS Xswp_60_0226={X 167.429794,Y 851.924683,Z 262.384491,A 175.758102,B 30.2117805,C 88.6917877,S 2,T 34,E1 5342.35693,E2 0.0,E3 0.0,E4 0.0,E5 0.0,E6 0.0}
DECL FDAT Fswp_60_0230={TOOL_NO 2,BASE_NO 2,IPO_FRAME #BASE,POINT2[] " "}
DECL PDAT PP_OLP38={VEL 100.0,ACC 100.0,APO_DIST 0.0}
DECL SPOT_TYPE SS_OLP8={GUN 1,PAIR #FIRST,RETR #OPN,CLO_TM 0,PGNO1 1,PRESS1 1.0,PGNO2 0,PRESS2 0.0}
DECL E6POS Xswp_60_0230={X 175.898499,Y 849.184998,Z 234.951797,A 176.958694,B 30.1404305,C 87.1446686,S 2,T 34,E1 5342.3501,E2 0.0,E3 0.0,E4 0.0,E5 0.0,E6 0.0}
DECL FDAT Fc_lx803={TOOL_NO 2,BASE_NO 2,IPO_FRAME #BASE,POINT2[] " "}
DECL PDAT PP_OLP39={VEL 100.0,ACC 100.0,APO_DIST 100.0,APO_MODE #CDIS}
DECL E6POS Xc_lx803={X 188.816101,Y 801.955383,Z 290.867401,A 175.750305,B 32.2371292,C 88.6945496,S 2,T 34,E1 5342.53711,E2 0.0,E3 0.0,E4 0.0,E5 0.0,E6 0.0}
DECL FDAT Fc_lx806={TOOL_NO 2,BASE_NO 2,IPO_FRAME #BASE,POINT2[] " "}
DECL PDAT PP_OLP42={VEL 100.0,ACC 100.0,APO_DIST 100.0,APO_MODE #CDIS}
DECL E6POS Xc_lx806={X 361.210114,Y 1274.42798,Z 281.714294,A -172.720001,B 54.0112801,C 88.4402008,S 2,T 34,E1 5392.10205,E2 0.0,E3 0.0,E4 0.0,E5 0.0,E6 0.0}
DECL FDAT Fc_lx801={TOOL_NO 2,BASE_NO 2,IPO_FRAME #BASE,POINT2[] " "}
DECL PDAT PP_OLP46={VEL 100.0,ACC 100.0,APO_DIST 100.0,APO_MODE #CDIS}
DECL E6POS Xc_lx801={X 383.558289,Y 1044.38599,Z -102.5317,A -173.268799,B 58.5109482,C 89.9160538,S 2,T 34,E1 5405.94385,E2 0.0,E3 0.0,E4 0.0,E5 0.0,E6 0.0}
DECL FDAT Fc_lx802={TOOL_NO 2,BASE_NO 2,IPO_FRAME #BASE,POINT2[] " "}
DECL PDAT PP_OLP47={VEL 100.0,ACC 100.0,APO_DIST 100.0,APO_MODE #CDIS}
DECL E6POS Xc_lx802={X 397.393188,Y 800.022827,Z -77.9418869,A -173.666306,B 52.2213898,C 91.9822769,S 2,T 34,E1 5405.94482,E2 0.0,E3 0.0,E4 0.0,E5 0.0,E6 0.0}
DECL FDAT Fc_lx800={TOOL_NO 2,BASE_NO 2,IPO_FRAME #BASE,POINT2[] " "}
DECL PDAT PP_OLP48={VEL 100.0,ACC 100.0,APO_DIST 100.0,APO_MODE #CDIS}
DECL E6POS Xc_lx800={X 347.276215,Y 816.817078,Z -64.3575897,A -174.908096,B 38.1721382,C 90.4691467,S 2,T 34,E1 5405.94482,E2 0.0,E3 0.0,E4 0.0,E5 0.0,E6 0.0}
DECL FDAT Fc_lx799={TOOL_NO 2,BASE_NO 2,IPO_FRAME #BASE,POINT2[] " "}
DECL PDAT PP_OLP49={VEL 100.0,ACC 100.0,APO_DIST 100.0,APO_MODE #CDIS}
DECL E6POS Xc_lx799={X 226.790405,Y 813.854309,Z -78.1323929,A -177.653397,B 32.0375519,C 88.8633804,S 2,T 34,E1 5405.94482,E2 0.0,E3 0.0,E4 0.0,E5 0.0,E6 0.0}
DECL FDAT Fc_lx798={TOOL_NO 2,BASE_NO 2,IPO_FRAME #BASE,POINT2[] " "}
DECL PDAT PP_OLP50={VEL 100.0,ACC 100.0,APO_DIST 100.0,APO_MODE #CDIS}
DECL E6POS Xc_lx798={X 230.175797,Y 791.29541,Z 90.7611008,A -176.350693,B -14.9320898,C 88.9359665,S 2,T 34,E1 5405.94482,E2 0.0,E3 0.0,E4 0.0,E5 0.0,E6 0.0}
DECL FDAT Fswp_60_0236={TOOL_NO 2,BASE_NO 2,IPO_FRAME #BASE,POINT2[] " "}
DECL PDAT PP_OLP51={VEL 100.0,ACC 100.0,APO_DIST 0.0}
DECL SPOT_TYPE SS_OLP9={GUN 1,PAIR #FIRST,RETR #OPN,CLO_TM 0,PGNO1 1,PRESS1 1.0,PGNO2 0,PRESS2 0.0}
DECL E6POS Xswp_60_0236={X 213.391998,Y 837.47467,Z 137.100296,A -176.395996,B -24.4397507,C 91.5723572,S 2,T 34,E1 5405.95215,E2 0.0,E3 0.0,E4 0.0,E5 0.0,E6 0.0}
DECL FDAT Fswp_60_0246={TOOL_NO 2,BASE_NO 2,IPO_FRAME #BASE,POINT2[] " "}
DECL SPOT_TYPE SS_OLP10={GUN 1,PAIR #FIRST,RETR #OPN,CLO_TM 0,PGNO1 1,PRESS1 1.0,PGNO2 0,PRESS2 0.0}
DECL E6POS Xswp_60_0246={X 199.1297,Y 837.23938,Z -25.1585503,A -177.183304,B 10.6243,C 88.9206238,S 2,T 34,E1 5405.94287,E2 0.0,E3 0.0,E4 0.0,E5 0.0,E6 0.0}
DECL FDAT Fswp_60_0256={TOOL_NO 2,BASE_NO 2,IPO_FRAME #BASE,POINT2[] " "}
DECL SPOT_TYPE SS_OLP11={GUN 1,PAIR #FIRST,RETR #OPN,CLO_TM 0,PGNO1 1,PRESS1 1.0,PGNO2 0,PRESS2 0.0}
DECL E6POS Xswp_60_0256={X 261.304108,Y 833.392395,Z -121.913101,A -179.192093,B 38.5857811,C 88.7741089,S 2,T 34,E1 5405.81104,E2 0.0,E3 0.0,E4 0.0,E5 0.0,E6 0.0}
DECL FDAT Fc_lx813={TOOL_NO 2,BASE_NO 2,IPO_FRAME #BASE,POINT2[] " "}
DECL PDAT PP_OLP57={VEL 100.0,ACC 100.0,APO_DIST 100.0,APO_MODE #CDIS}
DECL E6POS Xc_lx813={X 407.447388,Y 819.060486,Z -112.462898,A 179.922501,B 56.4042511,C 86.032753,S 2,T 34,E1 5368.32178,E2 0.0,E3 0.0,E4 0.0,E5 0.0,E6 0.0}
DECL FDAT Fc_lx814={TOOL_NO 2,BASE_NO 2,IPO_FRAME #BASE,POINT2[] " "}
DECL PDAT PP_OLP58={VEL 100.0,ACC 100.0,APO_DIST 100.0,APO_MODE #CDIS}
DECL E6POS Xc_lx814={X 262.36261,Y 1480.59204,Z -64.9219971,A 174.308899,B 60.7039986,C 78.5164566,S 2,T 34,E1 5359.85303,E2 0.0,E3 0.0,E4 0.0,E5 0.0,E6 0.0}
DECL FDAT Fc_lx817={TOOL_NO 2,BASE_NO 2,IPO_FRAME #BASE,POINT2[] " "}
DECL PDAT PP_OLP59={VEL 100.0,ACC 100.0,APO_DIST 100.0,APO_MODE #CDIS}
DECL E6POS Xc_lx817={X 1142.85999,Y 1324.38098,Z 187.560699,A -0.147523597,B 11.5094099,C -87.7053528,S 2,T 2,E1 6214.02979,E2 0.0,E3 0.0,E4 0.0,E5 0.0,E6 0.0}
DECL FDAT Fc_lx816={TOOL_NO 2,BASE_NO 2,IPO_FRAME #BASE,POINT2[] " "}
DECL PDAT PP_OLP60={VEL 100.0,ACC 100.0,APO_DIST 20.0,APO_MODE #CDIS}
DECL E6POS Xc_lx816={X 1124.91003,Y 804.700073,Z 168.560806,A -0.147076294,B 11.5091105,C -87.7059021,S 2,T 2,E1 6214.03223,E2 0.0,E3 0.0,E4 0.0,E5 0.0,E6 0.0}
DECL FDAT Fc_lx815={TOOL_NO 2,BASE_NO 2,IPO_FRAME #BASE,POINT2[] " "}
DECL PDAT PP_OLP61={VEL 100.0,ACC 100.0,APO_DIST 20.0,APO_MODE #CDIS}
DECL E6POS Xc_lx815={X 1203.88,Y 787.201721,Z 140.274506,A 1.55256295,B 16.7296505,C -86.9592285,S 2,T 2,E1 6214.02979,E2 0.0,E3 0.0,E4 0.0,E5 0.0,E6 0.0}
DECL FDAT Fswp_60_0334={TOOL_NO 2,BASE_NO 2,IPO_FRAME #BASE,POINT2[] " "}
DECL PDAT PP_OLP62={VEL 100.0,ACC 100.0,APO_DIST 0.0}
DECL SPOT_TYPE SS_OLP12={GUN 1,PAIR #FIRST,RETR #OPN,CLO_TM 0,PGNO1 1,PRESS1 1.0,PGNO2 0,PRESS2 0.0}
DECL E6POS Xswp_60_0334={X 1203.11804,Y 822.041992,Z 66.6144791,A 1.92325699,B 27.3806801,C -89.0109329,S 2,T 2,E1 6214.02393,E2 0.0,E3 0.0,E4 0.0,E5 0.0,E6 0.0}
DECL FDAT Fswp_60_0342={TOOL_NO 2,BASE_NO 2,IPO_FRAME #BASE,POINT2[] " "}
DECL PDAT PP_OLP63={VEL 100.0,ACC 100.0,APO_DIST 0.0}
DECL SPOT_TYPE SS_OLP13={GUN 1,PAIR #FIRST,RETR #OPN,CLO_TM 0,PGNO1 1,PRESS1 1.0,PGNO2 0,PRESS2 0.0}
DECL E6POS Xswp_60_0342={X 1346.99805,Y 823.695007,Z 68.5146713,A 0.944778502,B 30.4541607,C -90.6848526,S 2,T 2,E1 6214.0249,E2 0.0,E3 0.0,E4 0.0,E5 0.0,E6 0.0}
DECL FDAT Fc_lx820={TOOL_NO 2,BASE_NO 2,IPO_FRAME #BASE,POINT2[] " "}
DECL PDAT PP_OLP66={VEL 100.0,ACC 100.0,APO_DIST 100.0,APO_MODE #CDIS}
DECL E6POS Xc_lx820={X 1228.98096,Y 787.197693,Z 92.421402,A 2.18218207,B 27.3218307,C -86.7221375,S 2,T 2,E1 6214.02979,E2 0.0,E3 0.0,E4 0.0,E5 0.0,E6 0.0}
DECL FDAT Fc_lx822={TOOL_NO 2,BASE_NO 2,IPO_FRAME #BASE,POINT2[] " "}
DECL PDAT PP_OLP67={VEL 100.0,ACC 100.0,APO_DIST 25.0,APO_MODE #CDIS}
DECL E6POS Xc_lx822={X 1167.49597,Y 1329.48999,Z 729.390381,A -1.61207795,B -54.9786491,C -88.5424576,S 2,T 2,E1 6214.0332,E2 0.0,E3 0.0,E4 0.0,E5 0.0,E6 0.0}
DECL FDAT Fc_lx823={TOOL_NO 2,BASE_NO 2,IPO_FRAME #BASE,POINT2[] " "}
DECL PDAT PP_OLP68={VEL 100.0,ACC 100.0,APO_DIST 100.0,APO_MODE #CDIS}
DECL E6POS Xc_lx823={X 1190.40796,Y 826.939087,Z 711.113098,A -3.67346191,B -62.9607811,C -86.2920532,S 2,T 2,E1 6214.02979,E2 0.0,E3 0.0,E4 0.0,E5 0.0,E6 0.0}
DECL FDAT Fc_lx821={TOOL_NO 2,BASE_NO 2,IPO_FRAME #BASE,POINT2[] " "}
DECL PDAT PP_OLP69={VEL 100.0,ACC 100.0,APO_DIST 100.0,APO_MODE #CDIS}
DECL E6POS Xc_lx821={X 1348.82495,Y 821.645508,Z 707.689514,A -2.32652497,B -37.4837303,C -87.1951599,S 2,T 2,E1 6214.03223,E2 0.0,E3 0.0,E4 0.0,E5 0.0,E6 0.0}
DECL FDAT Fswp_60_0394={TOOL_NO 2,BASE_NO 2,IPO_FRAME #BASE,POINT2[] " "}
DECL PDAT PP_OLP70={VEL 100.0,ACC 100.0,APO_DIST 0.0}
DECL SPOT_TYPE SS_OLP14={GUN 1,PAIR #FIRST,RETR #OPN,CLO_TM 0,PGNO1 1,PRESS1 1.0,PGNO2 0,PRESS2 0.0}
DECL E6POS Xswp_60_0394={X 1413.724,Y 833.93103,Z 642.382019,A -1.02669001,B -16.5625191,C -87.5924072,S 2,T 2,E1 6214.02393,E2 0.0,E3 0.0,E4 0.0,E5 0.0,E6 0.0}
DECL FDAT Fc_lx824={TOOL_NO 2,BASE_NO 2,IPO_FRAME #BASE,POINT2[] " "}
DECL PDAT PP_OLP71={VEL 100.0,ACC 100.0,APO_DIST 100.0,APO_MODE #CDIS}
DECL E6POS Xc_lx824={X 1389.51404,Y 821.552917,Z 647.447876,A -1.545421,B -22.6872101,C -87.5638733,S 2,T 2,E1 6214.02979,E2 0.0,E3 0.0,E4 0.0,E5 0.0,E6 0.0}
DECL FDAT Fswp_60_0396={TOOL_NO 2,BASE_NO 2,IPO_FRAME #BASE,POINT2[] " "}
DECL PDAT PP_OLP72={VEL 100.0,ACC 100.0,APO_DIST 0.0}
DECL SPOT_TYPE SS_OLP15={GUN 1,PAIR #FIRST,RETR #OPN,CLO_TM 0,PGNO1 1,PRESS1 1.0,PGNO2 0,PRESS2 0.0}
DECL E6POS Xswp_60_0396={X 1386.58704,Y 831.857117,Z 677.264404,A -1.56504405,B -23.1201096,C -87.5573807,S 2,T 2,E1 6214.02979,E2 0.0,E3 0.0,E4 0.0,E5 0.0,E6 0.0}
DECL FDAT Fc_lx825={TOOL_NO 2,BASE_NO 2,IPO_FRAME #BASE,POINT2[] " "}
DECL PDAT PP_OLP73={VEL 100.0,ACC 100.0,APO_DIST 100.0,APO_MODE #CDIS}
DECL E6POS Xc_lx825={X 1387.53699,Y 824.184326,Z 740.618713,A -1.64721096,B -24.80303,C -87.522171,S 2,T 2,E1 6214.02979,E2 0.0,E3 0.0,E4 0.0,E5 0.0,E6 0.0}
DECL FDAT Fswp_60_0400={TOOL_NO 2,BASE_NO 2,IPO_FRAME #BASE,POINT2[] " "}
DECL PDAT PP_OLP74={VEL 100.0,ACC 100.0,APO_DIST 0.0}
DECL SPOT_TYPE SS_OLP16={GUN 1,PAIR #FIRST,RETR #OPN,CLO_TM 0,PGNO1 1,PRESS1 1.0,PGNO2 0,PRESS2 0.0}
DECL E6POS Xswp_60_0400={X 1414.49902,Y 836.641785,Z 743.982117,A -0.364520997,B -18.0130501,C -91.8461685,S 2,T 2,E1 6214.02979,E2 0.0,E3 0.0,E4 0.0,E5 0.0,E6 0.0}
DECL FDAT Fc_lx826={TOOL_NO 2,BASE_NO 2,IPO_FRAME #BASE,POINT2[] " "}
DECL PDAT PP_OLP75={VEL 100.0,ACC 100.0,APO_DIST 100.0,APO_MODE #CDIS}
DECL E6POS Xc_lx826={X 1388.27002,Y 820.920227,Z 742.32843,A -1.28494096,B -16.7925606,C -89.8897629,S 2,T 2,E1 6214.02979,E2 0.0,E3 0.0,E4 0.0,E5 0.0,E6 0.0}
DECL FDAT Fc_lx827={TOOL_NO 2,BASE_NO 2,IPO_FRAME #BASE,POINT2[] " "}
DECL PDAT PP_OLP76={VEL 100.0,ACC 100.0,APO_DIST 100.0,APO_MODE #CDIS}
DECL E6POS Xc_lx827={X 1348.91101,Y 818.656616,Z 707.930176,A -2.32552004,B -37.4811897,C -87.1952896,S 2,T 2,E1 6214.03223,E2 0.0,E3 0.0,E4 0.0,E5 0.0,E6 0.0}
DECL FDAT Fc_lx829={TOOL_NO 2,BASE_NO 2,IPO_FRAME #BASE,POINT2[] " "}
DECL PDAT PP_OLP78={VEL 100.0,ACC 100.0,APO_DIST 100.0,APO_MODE #CDIS}
DECL E6POS Xc_lx829={X 1192.28406,Y 826.407227,Z 711.405884,A -3.90112805,B -63.38591,C -86.059082,S 2,T 2,E1 6214.02979,E2 0.0,E3 0.0,E4 0.0,E5 0.0,E6 0.0}
DECL FDAT Fc_lx830={TOOL_NO 2,BASE_NO 2,IPO_FRAME #BASE,POINT2[] " "}
DECL PDAT PP_OLP79={VEL 100.0,ACC 100.0,APO_DIST 100.0,APO_MODE #CDIS}
DECL E6POS Xc_lx830={X 1161.22998,Y 1236.27002,Z 721.648376,A -4.67363214,B -62.0458603,C -85.0748291,S 2,T 2,E1 6214.03613,E2 0.0,E3 0.0,E4 0.0,E5 0.0,E6 0.0}
DECL FDAT Fc_lx770={TOOL_NO 2,BASE_NO 2,IPO_FRAME #BASE,POINT2[] " "}
DECL PDAT PP_OLP80={VEL 100.0,ACC 100.0,APO_DIST 100.0,APO_MODE #CDIS}
DECL E6POS Xc_lx770={X 1001.927,Y 1469.776,Z 577.685425,A -91.856308,B -67.3888321,C 12.5012503,S 2,T 2,E1 5891.69922,E2 0.0,E3 0.0,E4 0.0,E5 0.0,E6 0.0}
DECL BASIS_SUGG_T LAST_BASIS={POINT1[] "PS01010001              ",POINT2[] "PS01010001              ",CP_PARAMS[] "CPDAT0                  ",PTP_PARAMS[] "PDAT0                   ",CONT[] "                        ",CP_VEL[] "2.0                     ",PTP_VEL[] " 100                    ",SPL_NAME[] "S0                      "}
DECL SPOT_SUGG_T LAST_SPOT={GUN[] "2                       ",RETR_CMD[] "#OPN                    ",CHOISE[] "#FIRST                  ",CLO_TM[] "1                       ",PGNO1[] "1                       ",PRESS1[] "0                       ",PGNO2[] "1                       ",PRESS2[] "0                       ",SPOT_PARAMS[] "NORMAL                  "}
DECL E6POS XP3={X 1137.23804,Y 792.062988,Z 171.201294,A -0.147380903,B 11.5094604,C -87.7052231,S 2,T 2,E1 6214.02979,E2 0.0,E3 0.0,E4 0.0,E5 0.0,E6 0.0}
DECL FDAT FP3={TOOL_NO 2,BASE_NO 2,IPO_FRAME #BASE,POINT2[] " ",TQ_STATE FALSE}
DECL PDAT PPDAT3={VEL 100.0,ACC 100.0,APO_DIST 100.0,APO_MODE #CDIS}
DECL E6POS XP7={X 222.348007,Y 799.210571,Z 13.5823097,A -177.042694,B 5.62783098,C 88.9293518,S 2,T 34,E1 5405.94482,E2 0.0,E3 0.0,E4 0.0,E5 0.0,E6 0.0}
DECL FDAT FP7={TOOL_NO 2,BASE_NO 2,IPO_FRAME #BASE,POINT2[] " ",TQ_STATE FALSE}
DECL PDAT PPDAT16={VEL 100.0,ACC 100.0,APO_DIST 2.0,APO_MODE #CDIS}
DECL PDAT PP_OLP86={VEL 100.0,ACC 100.0,APO_DIST 100.0,APO_MODE #CDIS}
DECL E6POS Xc_lx831={X 351.138306,Y 1379.03296,Z -103.602699,A -173.768906,B 61.3369598,C 85.3822708,S 2,T 34,E1 5405.94385,E2 0.0,E3 0.0,E4 0.0,E5 0.0,E6 0.0}
DECL FDAT Fc_lx831={TOOL_NO 2,BASE_NO 2,IPO_FRAME #BASE,POINT2[] " "}
DECL E6POS XP10={X 181.096893,Y 874.411621,Z 543.037903,A 178.1436,B -18.2273808,C 93.6572418,S 2,T 34,E1 5325.17285,E2 0.0,E3 0.0,E4 0.0,E5 0.0,E6 0.0}
DECL FDAT FP10={TOOL_NO 2,BASE_NO 2,IPO_FRAME #BASE,POINT2[] " ",TQ_STATE FALSE}
DECL PDAT PPDAT19={VEL 100.0,ACC 100.0,APO_DIST 100.0,APO_MODE #CDIS}
DECL PDAT PPDAT29={VEL 100.0,ACC 100.0,APO_DIST 100.0}
DECL E6POS XP22={X 1135.46594,Y 1324.38196,Z 186.560196,A -0.149021596,B 11.5121098,C -87.7051163,S 2,T 2,E1 6214.02881,E2 0.0,E3 0.0,E4 0.0,E5 0.0,E6 0.0}
DECL FDAT FP22={TOOL_NO 2,BASE_NO 2,IPO_FRAME #BASE,POINT2[] " ",TQ_STATE FALSE}
DECL PDAT PPDAT38={VEL 100.0,ACC 100.0,APO_DIST 20.0,APO_MODE #CDIS}
DECL E6POS XP24={X 1404.02502,Y 824.589111,Z 635.479675,A -1.386289,B -20.0821209,C -87.7755737,S 2,T 2,E1 6214.0332,E2 0.0,E3 0.0,E4 0.0,E5 0.0,E6 0.0}
DECL FDAT FP24={TOOL_NO 2,BASE_NO 2,IPO_FRAME #BASE,POINT2[] " ",TQ_STATE FALSE}
DECL PDAT PPDAT41={VEL 100.0,ACC 100.0,APO_DIST 10.0,APO_MODE #CDIS}
DECL PDAT PP_OLP88={VEL 100.0,ACC 100.0,APO_DIST 100.0,APO_MODE #CDIS}
DECL E6POS Xc_lx832={X 384.786285,Y 1136.39099,Z -119.928497,A 176.126694,B 62.8486404,C 80.9144135,S 2,T 34,E1 5359.84912,E2 0.0,E3 0.0,E4 0.0,E5 0.0,E6 0.0}
DECL FDAT Fc_lx832={TOOL_NO 2,BASE_NO 2,IPO_FRAME #BASE,POINT2[] " "}
DECL E6POS XP26={X 373.632599,Y 795.344116,Z 324.714386,A -179.101196,B 51.2975006,C 88.7150192,S 2,T 34,E1 5364.28711,E2 0.0,E3 0.0,E4 0.0,E5 0.0,E6 0.0}
DECL FDAT FP26={TOOL_NO 2,BASE_NO 2,IPO_FRAME #BASE,POINT2[] " ",TQ_STATE FALSE}
DECL PDAT PPDAT43={VEL 100.0,ACC 100.0,APO_DIST 100.0,APO_MODE #CDIS}
DECL PDAT PPDAT44={VEL 100.0,ACC 100.0,APO_DIST 100.0}
DECL E6POS XP28={X 231.731903,Y 827.260315,Z 539.866089,A -174.169601,B -19.2986698,C 92.3134537,S 2,T 34,E1 5325.17285,E2 0.0,E3 0.0,E4 0.0,E5 0.0,E6 0.0}
DECL FDAT FP28={TOOL_NO 2,BASE_NO 2,IPO_FRAME #BASE,POINT2[] " ",TQ_STATE FALSE}
DECL PDAT PPDAT45={VEL 100.0,ACC 100.0,APO_DIST 20.0,APO_MODE #CDIS}
DECL PDAT PP_OLP92={VEL 75.0,ACC 75.0,APO_DIST 0.0}
DECL PDAT PP_OLP93={VEL 100.0,ACC 100.0,APO_DIST 100.0,APO_MODE #CDIS}
DECL E6POS Xc_lx836={X 194.993393,Y 818.700989,Z 390.977814,A -179.958496,B 3.35912395,C 89.4341125,S 2,T 34,E1 5344.41309,E2 0.0,E3 0.0,E4 0.0,E5 0.0,E6 0.0}
DECL FDAT Fc_lx836={TOOL_NO 2,BASE_NO 2,IPO_FRAME #BASE,POINT2[] " "}
DECL PDAT PP_OLP94={VEL 100.0,ACC 100.0,APO_DIST 100.0,APO_MODE #CDIS}
DECL E6POS Xc_lx837={X 153.897903,Y 821.798218,Z 298.17099,A 176.825195,B 14.57022,C 87.8231201,S 2,T 34,E1 5341.86377,E2 0.0,E3 0.0,E4 0.0,E5 0.0,E6 0.0}
DECL FDAT Fc_lx837={TOOL_NO 2,BASE_NO 2,IPO_FRAME #BASE,POINT2[] " "}
DECL PDAT PP_OLP95={VEL 100.0,ACC 100.0,APO_DIST 0.0}
DECL PDAT PP_OLP96={VEL 100.0,ACC 100.0,APO_DIST 100.0,APO_MODE #CDIS}
DECL E6POS Xc_lx838={X 174.025299,Y 840.041382,Z 298.2099,A 175.758408,B 30.2116108,C 88.691597,S 2,T 34,E1 5342.35498,E2 0.0,E3 0.0,E4 0.0,E5 0.0,E6 0.0}
DECL FDAT Fc_lx838={TOOL_NO 2,BASE_NO 2,IPO_FRAME #BASE,POINT2[] " "}
DECL PDAT PP_OLP97={VEL 100.0,ACC 100.0,APO_DIST 0.0}
DECL PDAT PPDAT63={VEL 100.0,ACC 100.0,APO_DIST 100.0}
DECL PDAT PPDAT64={VEL 100.0,ACC 100.0,APO_DIST 100.0}
DECL PDAT PPDAT65={VEL 100.0,ACC 100.0,APO_DIST 100.0}
DECL PDAT PPDAT66={VEL 100.0,ACC 100.0,APO_DIST 100.0}
DECL PDAT PP_OLP98={VEL 100.0,ACC 100.0,APO_DIST 0.0}
DECL PDAT PPDAT67={VEL 100.0,ACC 100.0,APO_DIST 100.0}
DECL PDAT PPDAT68={VEL 100.0,ACC 100.0,APO_DIST 100.0}
DECL PDAT PPDAT69={VEL 100.0,ACC 100.0,APO_DIST 100.0}
DECL PDAT PPDAT70={VEL 100.0,ACC 100.0,APO_DIST 100.0}
DECL PDAT PP_OLP99={VEL 100.0,ACC 100.0,APO_DIST 0.0}
DECL PDAT PPDAT71={VEL 100.0,ACC 100.0,APO_DIST 100.0}
DECL PDAT PPDAT72={VEL 100.0,ACC 100.0,APO_DIST 100.0}
DECL PDAT PPDAT73={VEL 100.0,ACC 100.0,APO_DIST 100.0,APO_MODE #CDIS}
DECL E6POS XP53={X -935.189026,Y 2849.75806,Z -566.933594,A 111.187798,B -1.17289698,C -11.4574003,S 2,T 42,E1 4076.1311,E2 0.0,E3 0.0,E4 0.0,E5 0.0,E6 0.0}
DECL FDAT FP53={TOOL_NO 2,BASE_NO 2,IPO_FRAME #BASE,POINT2[] " ",TQ_STATE FALSE}
DECL PDAT PPDAT74={VEL 100.0,ACC 100.0,APO_DIST 100.0,APO_MODE #CDIS}
DECL E6POS XP54={X -102.170502,Y 2558.13306,Z -180.740906,A -90.9388123,B -6.38708687,C 25.6022091,S 2,T 2,E1 5073.56494,E2 0.0,E3 0.0,E4 0.0,E5 0.0,E6 0.0}
DECL FDAT FP54={TOOL_NO 2,BASE_NO 2,IPO_FRAME #BASE,POINT2[] " ",TQ_STATE FALSE}
DECL PDAT PPDAT77={VEL 100.0,ACC 100.0,APO_DIST 100.0,APO_MODE #CDIS}
DECL E6POS XP57={X -102.170502,Y 2558.13306,Z -180.740906,A -90.9388123,B -6.38708687,C 25.6022091,S 2,T 2,E1 5073.56494,E2 0.0,E3 0.0,E4 0.0,E5 0.0,E6 0.0}
DECL FDAT FP57={TOOL_NO 2,BASE_NO 2,IPO_FRAME #BASE,POINT2[] " ",TQ_STATE FALSE}
DECL PDAT PPDAT79={VEL 100.0,ACC 100.0,APO_DIST 100.0,APO_MODE #CDIS}
DECL E6POS XP59={X -5345.3999,Y 3544.12305,Z -363.516602,A 5.63546085,B -3.36820292,C 7.47960901,S 2,T 11,E1 866.885376,E2 0.0,E3 0.0,E4 0.0,E5 0.0,E6 0.0}
DECL FDAT FP59={TOOL_NO 2,BASE_NO 2,IPO_FRAME #BASE,POINT2[] " ",TQ_STATE FALSE}
DECL PDAT PPDAT80={VEL 100.0,ACC 100.0,APO_DIST 100.0,APO_MODE #CDIS}
DECL E6POS XP60={X -4659.89111,Y 2710.31201,Z -340.069885,A -69.4399414,B -4.68788099,C 11.6254101,S 2,T 2,E1 866.890015,E2 0.0,E3 0.0,E4 0.0,E5 0.0,E6 0.0}
DECL FDAT FP60={TOOL_NO 2,BASE_NO 2,IPO_FRAME #BASE,POINT2[] " ",TQ_STATE FALSE}
DECL PDAT PP_OLP100={VEL 100.0,ACC 100.0,APO_DIST 100.0,APO_MODE #CDIS}
DECL E6POS Xc_lx839={X 27.3463402,Y 1154.65796,Z 231.319305,A -12.9030399,B -45.4888611,C -79.3028488,S 2,T 2,E1 5234.21484,E2 0.0,E3 0.0,E4 0.0,E5 0.0,E6 0.0}
DECL FDAT Fc_lx839={TOOL_NO 2,BASE_NO 2,IPO_FRAME #BASE,POINT2[] " "}
DECL PDAT PP_OLP101={VEL 100.0,ACC 100.0,APO_DIST 100.0,APO_MODE #CDIS}
DECL E6POS Xc_lx840={X 11.7854605,Y 813.580017,Z 253.7845,A -6.39366198,B -47.92033,C -88.1291733,S 2,T 2,E1 5234.21484,E2 0.0,E3 0.0,E4 0.0,E5 0.0,E6 0.0}
DECL FDAT Fc_lx840={TOOL_NO 2,BASE_NO 2,IPO_FRAME #BASE,POINT2[] " "}
DECL PDAT PPDAT81={VEL 100.0,ACC 100.0,APO_DIST 100.0,APO_MODE #CDIS}
DECL E6POS XP61={X 51.816391,Y 813.576172,Z 284.23999,A -6.01011276,B -35.9100418,C -88.6002579,S 2,T 2,E1 5234.21484,E2 0.0,E3 0.0,E4 0.0,E5 0.0,E6 0.0}
DECL FDAT FP61={TOOL_NO 2,BASE_NO 2,IPO_FRAME #BASE,POINT2[] " ",TQ_STATE FALSE}
DECL PDAT PPDAT82={VEL 100.0,ACC 100.0,APO_DIST 100.0}
DECL PDAT PPDAT83={VEL 100.0,ACC 100.0,APO_DIST 100.0}
DECL PDAT PPDAT84={VEL 100.0,ACC 100.0,APO_DIST 100.0,APO_MODE #CDIS}
DECL E6POS XP62={X 62.5355911,Y 815.795471,Z 342.454407,A -6.13695002,B -46.3835907,C -91.8145065,S 2,T 2,E1 5234.4292,E2 0.0,E3 0.0,E4 0.0,E5 0.0,E6 0.0}
DECL FDAT FP62={TOOL_NO 2,BASE_NO 2,IPO_FRAME #BASE,POINT2[] " ",TQ_STATE FALSE}
DECL PDAT PPDAT85={VEL 100.0,ACC 100.0,APO_DIST 100.0}
DECL PDAT PPDAT86={VEL 100.0,ACC 100.0,APO_DIST 100.0}
DECL E6POS Xswp_60_0212={X 118.467201,Y 854.133789,Z 446.298401,A 2.86171007,B -51.0715218,C -94.7051697,S 2,T 2,E1 5234.42822,E2 0.0,E3 0.0,E4 0.0,E5 0.0,E6 0.0}
DECL FDAT Fswp_60_0212={TOOL_NO 2,BASE_NO 2,IPO_FRAME #BASE,POINT2[] " "}
DECL PDAT PPDAT87={VEL 100.0,ACC 100.0,APO_DIST 100.0}
DECL PDAT PPDAT88={VEL 100.0,ACC 100.0,APO_DIST 100.0,APO_MODE #CDIS}
DECL E6POS XP65={X 62.533371,Y 815.795227,Z 342.451996,A -6.13714981,B -46.3839493,C -91.8143997,S 2,T 2,E1 5234.4292,E2 0.0,E3 0.0,E4 0.0,E5 0.0,E6 0.0}
DECL FDAT FP65={TOOL_NO 2,BASE_NO 2,IPO_FRAME #BASE,POINT2[] " ",TQ_STATE FALSE}
DECL PDAT PPDAT89={VEL 100.0,ACC 100.0,APO_DIST 100.0,APO_MODE #CDIS}
DECL E6POS XP66={X 11.7855597,Y 813.580017,Z 253.784302,A -6.39366388,B -47.92033,C -88.1291733,S 2,T 2,E1 5234.21484,E2 0.0,E3 0.0,E4 0.0,E5 0.0,E6 0.0}
DECL FDAT FP66={TOOL_NO 2,BASE_NO 2,IPO_FRAME #BASE,POINT2[] " ",TQ_STATE FALSE}
DECL PDAT PPDAT90={VEL 100.0,ACC 100.0,APO_DIST 100.0,APO_MODE #CDIS}
DECL E6POS XP67={X 27.3452702,Y 1154.65601,Z 231.321396,A -12.9031,B -45.4890709,C -79.3028717,S 2,T 2,E1 5234.21484,E2 0.0,E3 0.0,E4 0.0,E5 0.0,E6 0.0}
DECL FDAT FP67={TOOL_NO 2,BASE_NO 2,IPO_FRAME #BASE,POINT2[] " ",TQ_STATE FALSE}
DECL PDAT PPDAT91={VEL 100.0,ACC 100.0,APO_DIST 100.0,APO_MODE #CDIS}
DECL E6POS XP68={X 290.253815,Y 1238.10095,Z 562.768616,A 9.59664726,B -57.2444305,C -94.041481,S 2,T 2,E1 5125.17383,E2 0.0,E3 0.0,E4 0.0,E5 0.0,E6 0.0}
DECL FDAT FP68={TOOL_NO 2,BASE_NO 2,IPO_FRAME #BASE,POINT2[] " ",TQ_STATE FALSE}
DECL PDAT PPDAT92={VEL 100.0,ACC 100.0,APO_DIST 100.0,APO_MODE #CDIS}
DECL E6POS XP69={X 273.273499,Y 1177.81702,Z 538.151428,A -175.308304,B -34.2909012,C 91.4840698,S 2,T 2,E1 5125.1748,E2 0.0,E3 0.0,E4 0.0,E5 0.0,E6 0.0}
DECL FDAT FP69={TOOL_NO 2,BASE_NO 2,IPO_FRAME #BASE,POINT2[] " ",TQ_STATE FALSE}
DECL PDAT PPDAT94={VEL 100.0,ACC 100.0,APO_DIST 100.0,APO_MODE #CDIS}
DECL E6POS XP71={X 224.162598,Y 1533.74402,Z 228.679398,A -77.3140411,B -57.1955719,C 4.26798487,S 2,T 2,E1 5073.56494,E2 0.0,E3 0.0,E4 0.0,E5 0.0,E6 0.0}
DECL FDAT FP71={TOOL_NO 2,BASE_NO 2,IPO_FRAME #BASE,POINT2[] " ",TQ_STATE FALSE}
DECL PDAT PP_OLP102={VEL 100.0,ACC 100.0,APO_DIST 0.0}
DECL PDAT PP_OLP103={VEL 100.0,ACC 100.0,APO_DIST 0.0}
DECL E6POS Xswp_60_0336={X 1240.979,Y 823.661011,Z 66.0155869,A 0.71519351,B 31.2928905,C -90.0658569,S 2,T 2,E1 6214.02002,E2 0.0,E3 0.0,E4 0.0,E5 0.0,E6 0.0}
DECL FDAT Fswp_60_0336={TOOL_NO 2,BASE_NO 2,IPO_FRAME #BASE,POINT2[] " "}
DECL PDAT PP_OLP104={VEL 100.0,ACC 100.0,APO_DIST 0.0}
DECL PDAT PP_OLP105={VEL 100.0,ACC 100.0,APO_DIST 0.0}
DECL E6POS Xswp_60_0338={X 1275.65601,Y 822.661621,Z 65.4634323,A 1.55081499,B 26.3931007,C -90.0217972,S 2,T 2,E1 6214.021,E2 0.0,E3 0.0,E4 0.0,E5 0.0,E6 0.0}
DECL FDAT Fswp_60_0338={TOOL_NO 2,BASE_NO 2,IPO_FRAME #BASE,POINT2[] " "}
DECL E6POS Xswp_60_0208={X 173.335602,Y 857.06543,Z 445.694489,A 2.3256681,B -45.8590508,C -94.2442627,S 2,T 2,E1 5234.4248,E2 0.0,E3 0.0,E4 0.0,E5 0.0,E6 0.0}
DECL FDAT Fswp_60_0208={TOOL_NO 2,BASE_NO 2,IPO_FRAME #BASE,POINT2[] " ",TQ_STATE FALSE}
DECL E6POS Xswp_60_0204={X 219.412598,Y 876.562622,Z 536.998474,A -179.878494,B -18.7035408,C 92.4623871,S 2,T 34,E1 5325.1792,E2 0.0,E3 0.0,E4 0.0,E5 0.0,E6 0.0}
DECL FDAT Fswp_60_0204={TOOL_NO 2,BASE_NO 2,IPO_FRAME #BASE,POINT2[] " ",TQ_STATE FALSE}
DECL E6POS Xswp_60_0238={X 223.714096,Y 833.494324,Z 99.323822,A -176.048401,B -26.75214,C 88.2412109,S 2,T 34,E1 5405.94092,E2 0.0,E3 0.0,E4 0.0,E5 0.0,E6 0.0}
DECL FDAT Fswp_60_0238={TOOL_NO 2,BASE_NO 2,IPO_FRAME #BASE,POINT2[] " ",TQ_STATE FALSE}
DECL E6POS Xswp_60_0240={X 220.955597,Y 835.205017,Z 80.2341766,A -175.876694,B -31.5127106,C 88.1577835,S 2,T 34,E1 5405.93896,E2 0.0,E3 0.0,E4 0.0,E5 0.0,E6 0.0}
DECL FDAT Fswp_60_0240={TOOL_NO 2,BASE_NO 2,IPO_FRAME #BASE,POINT2[] " ",TQ_STATE FALSE}
DECL E6POS Xswp_60_0242={X 215.938797,Y 836.161621,Z 33.9351883,A -176.220505,B -21.63727,C 88.2889633,S 2,T 34,E1 5405.94189,E2 0.0,E3 0.0,E4 0.0,E5 0.0,E6 0.0}
DECL FDAT Fswp_60_0242={TOOL_NO 2,BASE_NO 2,IPO_FRAME #BASE,POINT2[] " ",TQ_STATE FALSE}
DECL E6POS Xswp_60_0244={X 209.4095,Y 833.383728,Z 5.23500776,A -176.873795,B 0.81782341,C 88.4093704,S 2,T 34,E1 5405.94092,E2 0.0,E3 0.0,E4 0.0,E5 0.0,E6 0.0}
DECL FDAT Fswp_60_0244={TOOL_NO 2,BASE_NO 2,IPO_FRAME #BASE,POINT2[] " ",TQ_STATE FALSE}
DECL E6POS Xswp_60_0248={X 190.353104,Y 835.066528,Z -51.7266006,A -177.317001,B 17.4398403,C 88.8883133,S 2,T 34,E1 5405.94092,E2 0.0,E3 0.0,E4 0.0,E5 0.0,E6 0.0}
DECL FDAT Fswp_60_0248={TOOL_NO 2,BASE_NO 2,IPO_FRAME #BASE,POINT2[] " ",TQ_STATE FALSE}
DECL E6POS Xswp_60_0250={X 181.176102,Y 836.54657,Z -90.4182129,A -177.352295,B 21.6734104,C 88.8233871,S 2,T 34,E1 5405.94092,E2 0.0,E3 0.0,E4 0.0,E5 0.0,E6 0.0}
DECL FDAT Fswp_60_0250={TOOL_NO 2,BASE_NO 2,IPO_FRAME #BASE,POINT2[] " ",TQ_STATE FALSE}
DECL E6POS Xswp_60_0252={X 198.7173,Y 838.126587,Z -103.778503,A -177.683105,B 33.3631706,C 88.7304077,S 2,T 34,E1 5405.94189,E2 0.0,E3 0.0,E4 0.0,E5 0.0,E6 0.0}
DECL FDAT Fswp_60_0252={TOOL_NO 2,BASE_NO 2,IPO_FRAME #BASE,POINT2[] " ",TQ_STATE FALSE}
DECL E6POS Xswp_60_0254={X 218.711594,Y 833.941895,Z -110.274101,A 179.148804,B 33.3342209,C 88.6294327,S 2,T 34,E1 5405.94189,E2 0.0,E3 0.0,E4 0.0,E5 0.0,E6 0.0}
DECL FDAT Fswp_60_0254={TOOL_NO 2,BASE_NO 2,IPO_FRAME #BASE,POINT2[] " ",TQ_STATE FALSE}
DECL E6POS Xswp_60_0258={X 294.644989,Y 833.254578,Z -121.963699,A 178.945496,B 48.5281906,C 88.5373383,S 2,T 34,E1 5405.81201,E2 0.0,E3 0.0,E4 0.0,E5 0.0,E6 0.0}
DECL FDAT Fswp_60_0258={TOOL_NO 2,BASE_NO 2,IPO_FRAME #BASE,POINT2[] " ",TQ_STATE FALSE}
DECL E6POS Xswp_60_0260={X 329.423096,Y 833.599976,Z -122.690903,A -179.874207,B 47.4368706,C 88.7545319,S 2,T 34,E1 5405.81299,E2 0.0,E3 0.0,E4 0.0,E5 0.0,E6 0.0}
DECL FDAT Fswp_60_0260={TOOL_NO 2,BASE_NO 2,IPO_FRAME #BASE,POINT2[] " ",TQ_STATE FALSE}
DECL E6POS Xswp_60_0332={X 1168.04102,Y 825.248291,Z 66.2790298,A 2.18056107,B 27.3222103,C -88.9835587,S 2,T 2,E1 6214.02197,E2 0.0,E3 0.0,E4 0.0,E5 0.0,E6 0.0}
DECL FDAT Fswp_60_0332={TOOL_NO 2,BASE_NO 2,IPO_FRAME #BASE,POINT2[] " ",TQ_STATE FALSE}
DECL E6POS Xswp_60_0340={X 1311.64294,Y 819.853516,Z 67.2476273,A 1.62332404,B 25.96632,C -90.0339432,S 2,T 2,E1 6214.01807,E2 0.0,E3 0.0,E4 0.0,E5 0.0,E6 0.0}
DECL FDAT Fswp_60_0340={TOOL_NO 2,BASE_NO 2,IPO_FRAME #BASE,POINT2[] " ",TQ_STATE FALSE}
DECL E6POS XP72={X -6762.21094,Y 2715.22705,Z -286.167999,A -1.43572199,B 5.65468884,C -0.0242798794,S 2,T 3,E1 866.892273,E2 0.0,E3 0.0,E4 0.0,E5 0.0,E6 0.0}
DECL FDAT FP72={TOOL_NO 2,BASE_NO 2,IPO_FRAME #BASE,POINT2[] " ",TQ_STATE FALSE}
DECL PDAT PPDAT95={VEL 100.0,ACC 100.0,APO_DIST 100.0}
DECL E6POS XP73={X -6304.68994,Y 3423.53809,Z -312.228088,A 37.3947105,B 0.75025183,C 10.5158195,S 2,T 3,E1 866.892578,E2 0.0,E3 0.0,E4 0.0,E5 0.0,E6 0.0}
DECL FDAT FP73={TOOL_NO 2,BASE_NO 2,IPO_FRAME #BASE,POINT2[] " ",TQ_STATE FALSE}
DECL PDAT PPDAT96={VEL 100.0,ACC 100.0,APO_DIST 100.0,APO_MODE #CDIS}
DECL PDAT PP_OLP77={VEL 100.0,ACC 100.0,APO_DIST 0.0}
DECL E6POS Xswp_60_0395={X 1417.83997,Y 833.93103,Z 642.382019,A -1.02669001,B -16.5625191,C -87.5924072,S 2,T 2,E1 6214.02393,E2 0.0,E3 0.0,E4 0.0,E5 0.0,E6 0.0}
DECL FDAT Fswp_60_0395={TOOL_NO 2,BASE_NO 2,IPO_FRAME #BASE,POINT2[] " "}
DECL E6POS Xswp_60_0392={X 1435.37903,Y 833.928711,Z 639.846985,A -0.429616511,B -2.21859598,C -87.6905823,S 2,T 2,E1 6214.02393,E2 0.0,E3 0.0,E4 0.0,E5 0.0,E6 0.0}
DECL FDAT Fswp_60_0392={TOOL_NO 2,BASE_NO 2,IPO_FRAME #BASE,POINT2[] " ",TQ_STATE FALSE}
DECL PDAT PP_OLP81={VEL 100.0,ACC 100.0,APO_DIST 0.0}
DECL E6POS Xswp_60_0397={X 1386.58704,Y 831.857117,Z 681.666382,A -1.56504405,B -23.1201096,C -87.5573807,S 2,T 2,E1 6214.02979,E2 0.0,E3 0.0,E4 0.0,E5 0.0,E6 0.0}
DECL FDAT Fswp_60_0397={TOOL_NO 2,BASE_NO 2,IPO_FRAME #BASE,POINT2[] " "}
DECL E6POS Xswp_60_0398={X 1387.70203,Y 831.05603,Z 706.325012,A -1.56509304,B -23.1200008,C -87.5572891,S 2,T 2,E1 6214.02979,E2 0.0,E3 0.0,E4 0.0,E5 0.0,E6 0.0}
DECL FDAT Fswp_60_0398={TOOL_NO 2,BASE_NO 2,IPO_FRAME #BASE,POINT2[] " ",TQ_STATE FALSE}
ENDDAT
